DEF_AcqErr.IdXML		:=	'5';
DEF_AcqErr.TagXML		:=	7;

DEF_Prm_Pos.IdXML		:=	'5';
DEF_Prm_Pos.TagXML		:=	8;

DEF_Position.IdXML		:=	'5';
DEF_Position.TagXML		:=	1;

DEF_Rotation.IdXML		:=	'5';
DEF_Rotation.TagXML		:=	4;

DEF_Surv_rotation.IdXML	:=	'5';
DEF_Surv_rotation.TagXML:=	5;

DEF_Jog.IdXML			:=	'5';
DEF_Jog.TagXML			:=	9;

DEF_Home.IdXML			:=	'5';
DEF_Home.TagXML			:=	2;

DEF_Interlock.IdXML		:=	'0';
DEF_Interlock.TagXML		:=	5;

DEF_Asserv.IdXML		:=	'5';
DEF_Asserv.TagXML		:=	10;

DEF_Desasserv.IdXML		:=	'5';
DEF_Desasserv.TagXML	:=	11;

DEF_Reset.IdXML			:=	'5';
DEF_Reset.TagXML		:=	12;

DEF_Lag_Distance.IdXML	:=	'5';
DEF_Lag_Distance.TagXML:=	13;

DEF_Limite_Switch.IdXML	:=	'5';
DEF_Limite_Switch.TagXML:=	14;

(* réception ordres externes*)
RCP_Zero	:=	M_Zero;
RCP_Bias	:=	M_Bias;
RCP_Read_Error_Mat	:=	M_Read_Error_Mat;

(*calcul de position absolue du codeur*)
STATE_Pos_Abs_Codeur := F_ReadMotorAbsPosition(fScalingFactor := CONF_Scaling_Factor, dPositionFeedback := IN_Position_Codeur);

(*Calcul position relative + controle cohérence*)
IF OP_Position.Etape.2 OR OP_Balayage.Etape.2 OR OP_Balayage.Etape.7 OR OP_Balayage.Etape.9 THEN
	VAR_Ctrl_Cons_Ok := FALSE;
	IF ( PRM_NPoste < 0) OR (PRM_NPoste > 8) OR ( PRM_NRef < 0) OR (PRM_NRef > 8) THEN
		VAR_Ctrl_Cons_Ok := FALSE;
	ELSE
		IF (PRM_NPoste =	0) THEN
			VAR_pos_poste	:= 	0.0;
		ELSE
			VAR_pos_poste 	:= 	CONF_Pos_Poste[PRM_NPoste];
		END_IF
		IF (PRM_NRef = 0) THEN
			VAR_Pos_ref		:= 	0.0;
		ELSE
			VAR_Pos_ref		:=	CONF_Pos_Ref[PRM_Nref];
		END_IF
		VAR_cons_pos		:=	PRM_Position - Var_Pos_Poste + Var_Pos_Ref ;
		IF NOT CONF_Mvt_Lineaire THEN
			WHILE VAR_Cons_Pos > 360.0 DO
				VAR_cons_pos := VAR_cons_pos - 360;
			END_WHILE
			WHILE VAR_Cons_Pos < 0.0 DO
				VAR_cons_pos := VAR_cons_pos + 360;
			END_WHILE
			VAR_Ctrl_Cons_Ok		:=	TRUE;
		ELSE
			IF ((VAR_Cons_Pos >= CONF_Min_Pos) AND (VAR_Cons_Pos <= CONF_Max_Pos))
					OR ((CONF_Min_Pos = 0.0) AND (CONF_Max_Pos = 0.0)) THEN
				VAR_Ctrl_Cons_Ok		:=	TRUE;
			END_IF
		END_IF
	END_IF;
END_IF;

(*Calcul position par rapport au balayage*)
IF OP_Balayage.Etape.7 THEN
	VAR_Cons_Pos2 := VAR_cons_pos + PRM_Angle_Bal/2;
ELSIF OP_Balayage.Etape.9 THEN
	VAR_Cons_Pos2 := VAR_cons_pos - PRM_Angle_Bal/2;
ELSIF OP_Balayage.Etape.2 THEN
	IF NOT PRM_BalPos THEN
		VAR_Cons_Pos2 := VAR_cons_pos;
	ELSE
		VAR_Cons_Pos2 := VAR_cons_pos - PRM_Angle_Bal/2;
	END_IF
ELSIF  OP_Balayage.Etape.0 THEN
	VAR_Cons_Pos2 := VAR_cons_pos;
END_IF
IF OP_Balayage.Etape.7 OR OP_Balayage.Etape.9 OR OP_Balayage.Etape.2 OR OP_Balayage.Etape.0 THEN
	VAR_Ctrl_Cons_ok2		:=	FALSE;
	IF NOT CONF_Mvt_Lineaire THEN
		WHILE VAR_Cons_Pos2 > 360.0 DO
			VAR_Cons_Pos2 := VAR_Cons_Pos2 - 360;
		END_WHILE
		WHILE VAR_Cons_Pos2 < 0.0 DO
			VAR_Cons_Pos2 := VAR_Cons_Pos2 + 360;
		END_WHILE
		VAR_Ctrl_Cons_ok2		:=	TRUE;
	ELSE
		IF ((VAR_Cons_Pos2 >= CONF_Min_Pos) AND (VAR_Cons_Pos2 <= CONF_Max_Pos))
				OR ((CONF_Min_Pos = 0.0) AND (CONF_Max_Pos = 0.0)) THEN
			VAR_Ctrl_Cons_ok2		:=	TRUE;
		END_IF
	END_IF
END_IF

(*memorisation consigne de vitesse et conversion en deg/s si nécessaire*)
IF OP_Rotation.Etape.2 OR OP_Balayage.Etape.2 THEN
	IF CONF_Mvt_Lineaire THEN
		VAR_V_BalRot	:=	PRM_V_BalRot;
	ELSE
		VAR_V_BalRot	:=	(PRM_V_BalRot * 360) / 60;
	END_IF
END_IF;
IF CONF_Mvt_Lineaire THEN
	VAR_V_Pos			:=	PRM_V_Pos;
	VAR_V_Rattrapage	:=	CONF_V_Rattrapage;
ELSE
	VAR_V_Pos			:=	(PRM_V_Pos * 360) / 60;
	VAR_V_Rattrapage	:=	(CONF_V_Rattrapage * 360) / 60;
END_IF

(*analyse besoin rattrapage de jeu*)
IF OP_Position.Etape.6 AND CONF_Rattrapage THEN
	IF CONF_Mvt_Lineaire THEN
		VAR_Pos	:=	STATE_Pos;
	ELSIF CONF_Deploiement THEN
		VAR_Pos	:=	STATE_Pos_Dep;
	ELSE
		VAR_Pos	:=	STATE_Pos360;
	END_IF
	IF CONF_Mvt_Lineaire OR CONF_Deploiement THEN
		VAR_Rattrapage	:=	((VAR_Cons_Pos2 > VAR_Pos) AND CONF_Sens_Rattrapage)
							OR ((VAR_Cons_Pos2 < VAR_Pos) AND NOT CONF_Sens_Rattrapage);
	ELSE
		VAR_Pos		:=	VAR_Cons_Pos2 - VAR_Pos;
		WHILE VAR_Pos > 360.0 DO
			VAR_Pos := VAR_Pos - 360;
		END_WHILE
		WHILE VAR_Pos < 0.0 DO
			VAR_Pos := VAR_Pos + 360;
		END_WHILE
		VAR_Sens_Mvt	:=	(VAR_Pos < 180.0);
		VAR_Rattrapage	:=	(VAR_Sens_Mvt AND CONF_Sens_Rattrapage)
							OR (NOT VAR_Sens_Mvt AND NOT CONF_Sens_Rattrapage);
	END_IF
END_IF

(*Front montant et descendant du mode manuel*)
FD_Manual.CLK	:=	MANUAL;
FD_Manual();

(*Front  validation esclave*)
FD_Valid_Slave.CLK	:=	CO_Valid_Slave;
FD_Valid_Slave();
FP_Valid_Slave.CLK	:=	CO_Valid_Slave;
FP_Valid_Slave();

(*Couple - Mise à l'échelle*)
STATE_Torque	:=	IN_Torque / 10;
END_ACTION

END_FUNCTION_BLOCK

// ---- POUs/Composant/MVTS/FB_WritePosBias.TcPOU
FUNCTION_BLOCK FB_WritePosBias
(****************historique des versions*****************************)
(* Version 1-0 - HG - 	VERSION INIITIALE*)
(* Version 2-0 - HG - 	retour nouvelle valeur position bias
					fonction d'écriture d'une valeur de position bias données*)
(* Version 3-0 - HG - 	gestion maj position bias pour une position non nulle*)
(*************************************************************************)

(*Commande bExecute:
permet de mettre à jour le paramètre position bias de la tache NC pour que 
la position courante (IPosBias) corresponde à la position zéro (IPosZero)
la nouvelle valeur du Position Bias est renvoyée dans STATE_PosBias
*)
(*Commande bApply:
permet de mettre à jour le paramètre position bias de la tache NC
directement à une valeur donnée (IPosBias) 
*)
VAR_INPUT
	bExecute: 		BOOL;
	bApply:			BOOL;
	id: 				UINT;
	lPosBias: 		LREAL;
	IPosZero:		LREAL:=0.0;
END_VAR
VAR_OUTPUT
	bBusy: 			BOOL;
	bErr: 			BOOL;
	bDone: 			BOOL;
	STATE_PosBias:	LREAL;
END_VAR
VAR
	step: 			UINT;
	VAR_PosBias:	LREAL;
	R_TRIG0: 		R_TRIG;
	R_TRIG1: 		R_TRIG;
	ADSWRITE0: 	ADSWRITE;
	ADSREAD0:		ADSREAD;
END_VAR

CASE step OF

	0:	(*lancement*)
		R_TRIG0(CLK := bExecute);
		R_TRIG1(CLK := bApply);
		bBusy := FALSE;
		IF R_TRIG0.Q THEN
			ADSWRITE0(WRITE := FALSE);
			ADSREAD0(READ := FALSE);
			bDone := FALSE;
			bBusy := TRUE;
			bErr := FALSE;
			step := step + 1;
		END_IF
		IF R_TRIG1.Q THEN
			ADSWRITE0(WRITE := FALSE);
			ADSREAD0(READ := FALSE);
			bDone := FALSE;
			bBusy := TRUE;
			bErr := FALSE;
			step := 2;
			VAR_PosBias := lPosBias;
		END_IF

	1:	(*lecture Position bias courant*)
		ADSREAD0(
			NETID:= '',
			PORT:= 501,
			IDXGRP:= id,
			IDXOFFS:= 16#07,
			LEN:= SIZEOF(VAR_PosBias),
			DESTADDR:= ADR(VAR_PosBias),
			READ:= TRUE,
			TMOUT:= t#500ms,);
		IF NOT ADSREAD0.BUSY THEN
			IF ADSREAD0.ERR THEN
				bErr := TRUE;
				step := 0;
			ELSE
				step 			:= 	step + 1;
				VAR_PosBias	:=	VAR_PosBias - lPosBias + IPosZero;
			END_IF
		END_IF

	2:	(*écriture position bias*)
		ADSWRITE0(
			NETID:= '',
			PORT:= 501,
			IDXGRP:= id,
			IDXOFFS:= 16#07,
			LEN:= SIZEOF(VAR_PosBias),
			SRCADDR:= ADR(VAR_PosBias),
			WRITE:= TRUE,
			TMOUT:= t#500ms);
		IF NOT ADSWRITE0.BUSY THEN
			IF ADSWRITE0.ERR THEN
				bErr := TRUE;
			ELSE
				bDone := TRUE;
				STATE_PosBias	:=	VAR_PosBias;
			END_IF
			step := 0;
		END_IF

END_CASE

END_FUNCTION_BLOCK

// ---- POUs/Composant/MVTS/F_ReadMotorAbsPosition.TcPOU
FUNCTION F_ReadMotorAbsPosition : LREAL			(* Fonction qui permet de lire la position absolue du moteur à codeur absolu avec AX5000 *)
VAR_INPUT
	fScalingFactor						: LREAL;		(* facteur de mise à l'échelle, nb mm/inc voir System Manager *)
	dPositionFeedback					: DINT;			(* valeur de retour de position de l'AX5000 *)
END_VAR
VAR
	dNbTours							: DINT;			(* nombre de tours du codeur *)
	dNbInc								: DINT;			(* nombre d'inc sur le tour *)
END_VAR

dNbTours := SHR(dPositionFeedback, 20);	(* le nombre de tours est sur les 12 bits de poids fort *)
dNbInc := DINT_TO_DWORD(dPositionFeedback) AND 2#00000000000011111111111111111111;	(* le nombre d'inc est sur 20 bits *)
F_ReadMotorAbsPosition := (dNbTours * 1048576 * fScalingFactor) + (dNbInc * fScalingFactor);

END_FUNCTION

// ---- POUs/Composant/MVTS/BLOCK_MOTEUR_ATV_ETHERCAT.TcPOU
{attribute 'call_after_init'}
FUNCTION_BLOCK BLOCK_MOTEUR_ATV_ETHERCAT

(* Element rotatif consigne ana *)

(****************historique des versions*****************************)
(* Version 0-0 - HG - VERSION INIITIALE - basée sur BLOCK_MOTEUR_ATV*)
(* Version 0-1 - HG - Corrections suite débug HC*)
(*************************************************************************)

VAR_INPUT
	RESET:							BOOL;		(* Condition de réinitialisation de la fonction *)

	I_Valid_INPUT:					BOOL;		(*INPUT valide - données exploitables*)
	
	IN_WcState	 		AT %I*:		BOOL;		(*INPUT IO-link Data process*)
	IN_InfoDataState 	AT %I*:		UINT;		(*INPUT Device Slave State*)

	IN_Status			AT %I*:		UINT;		(* INPUT - Entrée statut variateur*)
	IN_Error			AT %I*:		UINT;		(* INPUT - Erreur*)
	
	OP_MVT:							BLOCK_G7;
	
	DEF_WcState:					PRCDEF;		(* Défaut données invalides - communication figée*)
	DEF_Slave:						PRCDEF;		(* Défaut esclave EtherCAT*)
	DEF_off_auto:					PRCDEF;		(* Défaut de rupture de la chaîne de sécurité*)
	DEF_Variateur:					PRCDEF;		(* Défaut indiquant que le variateur n'est pas ok*)

	PRM_Vitesse:					REAL;		(* Consigne vitesse moteur*)
	PRM_Rapport:					REAL;		(* Rapport chaine cinématique*)
	
	CO_On:							BOOL;		(* Marche moteur en automatique*)
END_VAR

VAR_OUTPUT
	OUT_Control		AT %Q*:			UINT;		(* OUTPUT - Sortie mode de controle*)
	OUT_Velocity	AT %Q*:			INT;		(* OUTPUT - Sortie consigne vitesse, attention sortie en rpm ex: moteur a Vnom 1500 rpm*)

	STATE_Ready:					BOOL; 		(* Moteur pret*)
	STATE_OFF:						BOOL;		(* Moteur à l'arrêt *)
	STATE_EC:						BOOL;		(* Asservissement en cours *)
	STATE_ON:						BOOL;		(* Moteur en marche  *)
	STATE_NOK:						BOOL;		(* Moteur en defaut  *)
	STATE_VIT:						REAL;		(* Vitesse appliquée *)
END_VAR

VAR
	VAR_Valid_Elmt:					BOOL;		(*données EtherCAT exploitables*)

	VAR_On:							BOOL;		(* variable intermédiaire de marche moteur*)
	
	VAR_IN_ReadyToSwitchOn:			BOOL;		(* En attente de l'alimentation de puissance=1*)
	VAR_IN_SwitchedOn:				BOOL;		(*Ready*)
	VAR_IN_OperationEnabled:		BOOL;		(*En fonctionnement*)
	VAR_IN_Fault:					BOOL;		(* error*)
	VAR_IN_VoltageEnabled:			BOOL;		(*Alim puissance présente *)
	VAR_IN_QuickStop:				BOOL;		(* Arret rapide =0*)		
	VAR_IN_SwitchOnDisabled:		BOOL;		(* Absence Alim puissance *)
	VAR_IN_Warning:					BOOL;		(* Alarme présente*)
	VAR_IN_Reserve1:				BOOL;
	VAR_IN_Remote:					BOOL;		(* Commande via bus de terrain*)
	VAR_IN_TargetReached:			BOOL;		(* Référence atteinte*)
	VAR_IN_InternalLimitActive:		BOOL;		(* Déppassement réf*)
	VAR_IN_Reserve2:				BOOL;
	VAR_IN_Reserve3:				BOOL;
	VAR_IN_Conf1:					BOOL;		(* Stop button*)
	VAR_IN_Conf2:					BOOL;		(*Sens de rotations*)
	VAR_Status_Code:				USINT;		(*1: not ready to switch on, 2: switch on disabled, 3: ready to switch on,
												4: switched on, 5: operation enabled, 6: quick stop active,
												7: fault reaction active, 8: fault*)														
	VAR_OUT_SwitchOn:				BOOL;		(*Contrôle du switch principal*)
	VAR_OUT_EnableVoltage:			BOOL;		(*Mise en puissance*)
	VAR_OUT_QuickStop:				BOOL;		(*Quick stop activé =0*)
	VAR_OUT_EnableOperation:		BOOL;		(*Commande activée =1*)
	VAR_OUT_Reserve1:				BOOL;
	VAR_OUT_Reserve2:				BOOL;
	VAR_OUT_Reserve3:				BOOL;
	VAR_OUT_FaultReset:				BOOL;		(*0 à 1 pour reset erreur si l'erreur n'est plus active*)
	VAR_OUT_Halt:					BOOL;		(*0= run demandé, 1=arrêt demandé*)
	VAR_OUT_Reserve4:				BOOL;
	VAR_OUT_Reserve5:				BOOL;
	VAR_OUT_Conf1:					BOOL;		(*C311 - Marche avant par défaut*)  (*0= Marche avant demandée, 1= marche arrière demandée*)
	VAR_OUT_Conf2:					BOOL;		(*C312 - Marche arrière par défaut*)
	VAR_OUT_Conf3:					BOOL;		(*C313*)
	VAR_OUT_Conf4:					BOOL;		(*C314*)
	VAR_OUT_Conf5:					BOOL;		(*C315*)
	
	TIMER_Reset:					TON;
	TIMER_Timeout_Fault:			TON;
END_VAR

VAR_INPUT PERSISTENT
	CONF_VMAX:					REAL;			(*Consigne vitesse max*)
	CONF_VMIN:					REAL;			(*Consigne vitesse min*)
	CONF_No_Safety_Auto:		BOOL:=FALSE;	(*Option de desactivation des conditions d'autorisation en mode automatique*)
	
	(*Entité*)
	IsComponent:		BOOL;			(*entité : assembly*)
	IdXML:			STRING;			(*nom entité : identifiant pour recherche dans dico*)
	TagXML:			UINT;			(*nom entité : identifiant pour recherche dans dico*)
	IdParent:			STRING;			(*MNEMO de l'appelant*)
	MNEMO:			STRING;			(*MNEMO de l'entité*)
END_VAR

IdXML:= '5';
TagXML:= 2;

DEF_OFF_AUTO.IdXML := '3';
DEF_OFF_AUTO.TagXML :=10;
DEF_Variateur.IdXML	:= '5';
DEF_Variateur.TagXML:= 15;
DEF_Slave.IdXML := '19';
DEF_Slave.TagXML := 2;
DEF_WcState.IdXML := '19';
DEF_WcState.TagXML := 1;

(*DEFAUTS ESCLAVE ETHERCAT*)
(*Défaut données invalides*)
DEF_WcState.CONDITION	:=	IN_WcState AND NOT I_Valid_INPUT;
DEF_WcState();
(*Défaut esclave etherCAT*)
DEF_Slave.CONDITION		:=	(IN_InfoDataState<>8) AND NOT I_Valid_INPUT;
DEF_Slave.VAL1			:=	UINT_TO_STRING(IN_InfoDataState);
DEF_Slave();

(*Données E/S valables*)
VAR_Valid_Elmt			:=	I_Valid_INPUT AND NOT DEF_WcState.DEF AND NOT DEF_Slave.DEF;

(*Réception status*)
VAR_IN_ReadyToSwitchOn		:=	IN_Status.0;
VAR_IN_SwitchedOn			:=	IN_Status.1;
VAR_IN_OperationEnabled		:=	IN_Status.2;
VAR_IN_Fault				:=	IN_Status.3;
VAR_IN_VoltageEnabled		:=	IN_Status.4;
VAR_IN_QuickStop			:=	IN_Status.5;
VAR_IN_SwitchOnDisabled		:=	IN_Status.6;
VAR_IN_Warning				:=	IN_Status.7;
VAR_IN_Reserve1				:=	IN_Status.8;
VAR_IN_Remote				:=	IN_Status.9;
VAR_IN_TargetReached		:=	IN_Status.10;
VAR_IN_InternalLimitActive	:=	IN_Status.11;
VAR_IN_Reserve2				:=	IN_Status.12;
VAR_IN_Reserve3				:=	IN_Status.13;
VAR_IN_Conf1				:=	IN_Status.14;
VAR_IN_Conf2				:=	IN_Status.15;

(*CODE STATUS*)
IF NOT VAR_IN_ReadyToSwitchOn AND NOT VAR_IN_SwitchedOn AND NOT VAR_IN_OperationEnabled AND NOT VAR_IN_Fault AND NOT VAR_IN_SwitchOnDisabled THEN
	VAR_Status_Code	:=	1;	(*Not ready to switch on*)
ELSIF NOT VAR_IN_ReadyToSwitchOn AND NOT VAR_IN_SwitchedOn AND NOT VAR_IN_OperationEnabled AND NOT VAR_IN_Fault AND VAR_IN_SwitchOnDisabled THEN
	VAR_Status_Code	:=	2;	(*Switch on disabled*)
ELSIF VAR_IN_ReadyToSwitchOn AND NOT VAR_IN_SwitchedOn AND NOT VAR_IN_OperationEnabled AND NOT VAR_IN_Fault AND VAR_IN_QuickStop AND NOT VAR_IN_SwitchOnDisabled THEN
	VAR_Status_Code	:=	3;	(*Ready to switch on*)
ELSIF VAR_IN_ReadyToSwitchOn AND VAR_IN_SwitchedOn AND NOT VAR_IN_OperationEnabled AND NOT VAR_IN_Fault AND VAR_IN_VoltageEnabled AND VAR_IN_QuickStop AND NOT VAR_IN_SwitchOnDisabled THEN
	VAR_Status_Code	:=	4;	(*Switched on*)
ELSIF VAR_IN_ReadyToSwitchOn AND VAR_IN_SwitchedOn AND VAR_IN_OperationEnabled AND NOT VAR_IN_Fault AND VAR_IN_VoltageEnabled AND VAR_IN_QuickStop AND NOT VAR_IN_SwitchOnDisabled THEN
	VAR_Status_Code	:=	5;	(*Operation enabled*)
ELSIF VAR_IN_ReadyToSwitchOn AND VAR_IN_SwitchedOn AND VAR_IN_OperationEnabled AND NOT VAR_IN_Fault AND VAR_IN_VoltageEnabled AND NOT VAR_IN_QuickStop AND NOT VAR_IN_SwitchOnDisabled THEN
	VAR_Status_Code	:=	6;	(*Quick stop active*)
ELSIF VAR_IN_ReadyToSwitchOn AND VAR_IN_SwitchedOn AND VAR_IN_OperationEnabled AND VAR_IN_Fault AND NOT VAR_IN_SwitchOnDisabled THEN
	VAR_Status_Code	:=	7;	(*Fault reaction active*)
ELSIF NOT VAR_IN_ReadyToSwitchOn AND NOT VAR_IN_SwitchedOn AND NOT VAR_IN_OperationEnabled AND VAR_IN_Fault AND NOT VAR_IN_SwitchOnDisabled THEN
	VAR_Status_Code	:=	8;	(*Fault*)
END_IF


(*Vérification consignes*)
IF	PRM_Vitesse > CONF_VMAX THEN
	PRM_Vitesse	:=	CONF_VMAX;
END_IF;

IF PRM_Vitesse < CONF_VMIN THEN
	PRM_Vitesse := CONF_VMIN;
END_IF


(*défaut desactivation automatique*)
DEF_off_auto.CONDITION	:=	(DEF_Variateur.DEF AND NOT OP_MVT.Etape.1 AND NOT OP_MVT.Etape.2 AND NOT OP_MVT.Etape.0)
							OR TIMER_Timeout_Fault.Q;
DEF_off_auto.DELAY		:=	T#0MS;
DEF_off_auto();

(*défaut du variateur*)
DEF_Variateur.CONDITION		:= 	VAR_IN_Fault OR VAR_IN_Warning;
DEF_Variateur.VAL1			:=	UINT_TO_STRING(IN_Error);
DEF_Variateur.DELAY			:= 	T#5MS;
DEF_Variateur();

(*Indicateur prêt*)
STATE_Ready		:=	VAR_Valid_Elmt;

(*gestion des sorties*)
VAR_On		:= 	CO_ON AND NOT RESET;

(*appel G7*)
ACT_MVT();


(*consigne vitesse*)
IF	STATE_ON AND (PRM_VITESSE<>STATE_VIT) THEN
	OUT_Velocity	:=	REAL_TO_INT(PRM_Vitesse*PRM_Rapport);
	STATE_VIT		:=	PRM_Vitesse;
ELSIF STATE_OFF THEN
	OUT_Velocity	:=	0;
	STATE_VIT		:=	0;
END_IF;

(*PILOTAGE MODE DE CONTROLE*)
VAR_OUT_Conf1		:=	FALSE;
VAR_OUT_Conf2		:=	FALSE;
VAR_OUT_Conf3		:=	FALSE;
VAR_OUT_Conf4		:=	FALSE;
VAR_OUT_Conf5		:=	FALSE;
VAR_OUT_Reserve1	:=	FALSE;
VAR_OUT_Reserve2	:=	FALSE;
VAR_OUT_Reserve3	:=	FALSE;
VAR_OUT_Reserve4	:=	FALSE;
VAR_OUT_Reserve5	:=	FALSE;

VAR_OUT_Halt		:=	FALSE;

VAR_OUT_FaultReset		:=	OP_MVT.Etape.2;
VAR_OUT_EnableVoltage	:=	OP_MVT.Etape.3 OR OP_MVT.Etape.4 OR OP_MVT.Etape.5 OR OP_MVT.Etape.6 OR OP_MVT.Etape.7;
VAR_OUT_SwitchOn		:=	OP_MVT.Etape.4 OR OP_MVT.Etape.5 OR OP_MVT.Etape.6 OR OP_MVT.Etape.7;
VAR_OUT_QuickStop		:=	OP_MVT.Etape.3 OR OP_MVT.Etape.4 OR OP_MVT.Etape.5 OR OP_MVT.Etape.6 OR OP_MVT.Etape.7;
VAR_OUT_EnableOperation	:=	OP_MVT.Etape.5 OR OP_MVT.Etape.6;
//VAR_OUT_Conf1			:=	OP_MVT.Etape.6 AND (PRM_Vitesse > 0.0);

//MEMCPY(ADR(OUT_Control),ADR(VAR_OUT_SwitchOn),16);
OUT_CONTROL.0:=VAR_OUT_SwitchOn;
OUT_CONTROL.1:=VAR_OUT_EnableVoltage;
OUT_CONTROL.2:=VAR_OUT_QuickStop;
IdXML:= '5';
TagXML:= 2;

DEF_OFF_AUTO.IdXML := '3';
DEF_OFF_AUTO.TagXML :=10;
(*DEF_MARCHE.IdXML := '3';
DEF_MARCHE.TagXML:=1;*)
DEF_Variateur.IdXML	:= '5';
DEF_Variateur.TagXML:= 15;
	
	
OUT_CONTROL.3:=VAR_OUT_EnableOperation;
OUT_CONTROL.4:=VAR_OUT_Reserve1;
OUT_CONTROL.5:=VAR_OUT_Reserve2;
OUT_CONTROL.6:=VAR_OUT_Reserve3;
OUT_CONTROL.7:=VAR_OUT_FaultReset;
OUT_CONTROL.8:=VAR_OUT_Halt;
OUT_CONTROL.9:=VAR_OUT_Reserve4;
OUT_CONTROL.10:=VAR_OUT_Reserve5;
OUT_CONTROL.11:=VAR_OUT_Conf1;
OUT_CONTROL.12:=VAR_OUT_Conf2;
OUT_CONTROL.13:=VAR_OUT_Conf3;
OUT_CONTROL.14:=VAR_OUT_Conf4;
OUT_CONTROL.15:=VAR_OUT_Conf5;


(*Gestion du TIMER RESET*)
Timer_reset.IN:=OP_MVT.Etape.2;
Timer_reset.PT:= T#2S;
Timer_reset();

(*Gestion du TIMER Timout reset*)
TIMER_Timeout_Fault.IN:=OP_MVT.Etape.1 OR OP_MVT.Etape.2;
TIMER_Timeout_Fault.PT:=T#7S;
TIMER_Timeout_Fault();

(*Indicateur defaut*)
STATE_NOK	:=	DEF_off_auto.DEF OR DEF_Variateur.DEF OR DEF_WcState.DEF OR DEF_Slave.DEF;
STATE_ON	:=	OP_MVT.Etape.6;
STATE_OFF	:=	OP_MVT.Etape.0;
STATE_EC	:=	NOT STATE_ON AND NOT STATE_OFF;

ACTION ACT_MVT:
OP_MVT(
	N_STEP_OP_OK:= 6,
	N_STEP_OP_NOK:= 0);

(*GRAFCET*)
(* initialisation du grafcet*)
IF 		OP_MVT.ETAPE = 0
		THEN
				OP_MVT.ETAPE.0 := TRUE;
(*repositionnement sur étape 0*)
ELSIF	(NOT VAR_On OR DEF_off_auto.DEF)
		AND NOT OP_MVT.Etape.6 AND NOT OP_MVT.Etape.7
		THEN
				OP_MVT.ETAPE := 0;			(*RAZ grafcet*)
				OP_MVT.ETAPE.0:=TRUE;
(*étape 0-1*)
ELSIF 	OP_MVT.ETAPE.0
		AND VAR_On
		THEN
				OP_MVT.ETAPE.1:=TRUE;
				OP_MVT.ETAPE.0:=FALSE;
(*étape 1-2 : Fault*)
ELSIF	OP_MVT.Etape.1
		AND (VAR_Status_Code = 8)
		THEN
				OP_MVT.ETAPE.2:=TRUE;
				OP_MVT.ETAPE.1:=FALSE;
(*étape 2-1 : reset fault*)
ELSIF	OP_MVT.Etape.2
		AND TIMER_Reset.Q
		THEN
				OP_MVT.ETAPE.1:=TRUE;
				OP_MVT.ETAPE.2:=FALSE;				
(*étape 1-3*)
ELSIF	OP_MVT.Etape.1
		AND (VAR_Status_Code >= 2)
		THEN
				OP_MVT.ETAPE.3:=TRUE;
				OP_MVT.ETAPE.1:=FALSE;		
(*étape 3-4*)
ELSIF	OP_MVT.Etape.3
		AND (VAR_Status_Code >= 3)
		THEN
				OP_MVT.ETAPE.4:=TRUE;
				OP_MVT.ETAPE.3:=FALSE;	
(*étape 4-5*)
ELSIF	OP_MVT.Etape.4
		AND (VAR_Status_Code = 4)
		THEN
				OP_MVT.ETAPE.5:=TRUE;
				OP_MVT.ETAPE.4:=FALSE;
(*étape 5-6*)
ELSIF	OP_MVT.Etape.5
		AND (VAR_Status_Code = 5)
		THEN
				OP_MVT.ETAPE.6:=TRUE;
				OP_MVT.ETAPE.5:=FALSE;
(*étape 6-7*)
ELSIF	OP_MVT.Etape.6
		AND (NOT VAR_On OR DEF_off_auto.DEF)
		THEN
				OP_MVT.ETAPE.7:=TRUE;
				OP_MVT.ETAPE.6:=FALSE;
(*étape 7-0*)
ELSIF	OP_MVT.Etape.7
		AND (VAR_Status_Code <> 5)
		THEN
				OP_MVT.ETAPE.0:=TRUE;
				OP_MVT.ETAPE.7:=FALSE;
END_IF

OP_MVT.POST();
END_ACTION

END_FUNCTION_BLOCK

// ---- POUs/Composant/POMPES/BLOCK_PPM_DEF.TcPOU
FUNCTION_BLOCK BLOCK_PPM_DEF

(* Gestion d'une pompe turbo ADIXEN avec controleur REMOTE*)
(* TYPE OBJET = POMPE TURBO*)

(****************historique des versions*****************************)

(* Version 1-0 - HG - VERSION INIITIALE - 7015*)
(* Version 2-0 - HG - 06/2011 - Adaptation pour journal des évènements externe*)

(*************************************************************************)

VAR_INPUT
	MANUAL:					BOOL;				(* Mode de pilotage manuel *)
	RESET:					BOOL;				(* Condition de réiinitialisation de la fonction *)
	WATER:					BOOL;				(*indication de refrodissement de la pompe ok*)

	DEF_Arret_Auto:			PRCDEF;		(*01 - défaut d'arrêt automatique de la pompe*)
	DEF_Marche_imposs:		PRCDEF;		(*02 - défaut de marche de la pompe turbo non autorisée*)
	DEF_Arret_imposs:		PRCDEF;		(*03 - défaut d'arrêt de la pompe turbo non autorisée*)
	DEF_On:					PRCDEF;		(*04 - défaut de marche de la pompe*)
	DEF_Off:				PRCDEF;		(*05 - défaut d'arrêt de la pompe*)
	DEF_Interne:			PRCDEF;		(*06 - défaut interne de la pompe*)

	CO_On:					BOOL;			(*demande de marche de la pompe en mode automatique généré par la fonction qui gère la pompe*)

	(*conditions d'autorisation*)
	EN_On_INT:					BOOL:= TRUE;	(*condition d'autorisation de marche et de standby de la pompe donnée par la fonction qui gère la pompe*)
	EN_Off_INT:					BOOL:= TRUE;	(*condition d'autorisation d'arrêt de la pompe donnée par la fonction qui gère la pompe*)
	EN_On_EXT:					BOOL:= TRUE;	(*condition d'autorisation de marche et de standby externe*)
	EN_Off_EXT:					BOOL:= TRUE;	(*condition d'autorisation d'arrêt de la pompe donnée par la fonction qui gère la pompe*)

	IN_On:						BOOL;			(*entrée TOR pompe en marche*)
	IN_Def:						BOOL;			(*entrée TOR pompe en défaut*)

	OUT_On:						BOOL;			(* Marche pompe *)
END_VAR

VAR_INPUT PERSISTENT
	CONF_Tim_Valid_On:			TIME:=T#0ms;	(*temporisation de validation du l'état STATE_OK*)
	CONF_Tim_Valid_Off:			TIME:=T#0ms;	(*temporisation de validation de l'état STATE_AR*)

	(*Entité*)
	IsComponent:		BOOL;			(*entité : composant*)
	IdXML:				STRING;			(*nom entité : identifiant pour recherche dans dico*)
	TagXML:				UINT;			(*nom entité : identifiant pour recherche dans dico*)
	IdParent:			STRING;			(*MNEMO de l'appelant*)
	MNEMO:				STRING;			(*MNEMO de l'entité*)
END_VAR

VAR_OUTPUT
	RQ_Cool:					BOOL;			(* Demande de refroidissement de la pompe turbo*)

	(*variable d'état d'autorisation*)
	AUTOR_On_IHM:				BOOL;			(*indique que la mise en marche de la pompe est autorisée en mode manuel depuis l'IHM*)
	AUTOR_Off_IHM:				BOOL;			(*indique que l'arrêt de la pompe est autorisée en mode manuel depuis l'IHM*)

	STATE_Ec:					BOOL;			(*indique que la pompe est en marche et n'a pas atteint sa vitesse*)
	STATE_On:					BOOL;			(*indique que la pompe est en marche et à atteint sa vitesse*)
	STATE_NOK:					BOOL;			(*indique la présence d'un défaut sur la pompe ou que l'ordre de marche a été refusé*)
	STATE_Off:					BOOL;			(*indique que la pompe est à l'arrêt*)
	STATE_Ihm:					USINT;			(*code d'état de la pompe*)
END_VAR

VAR
	TIMER_Valid_On:				TON;
	TIMER_Valid_Off:			TON;

	(* Variables demande en mode manuel*)
	M_On:						BOOL;			(* Ordre marche/arrêt de la  pompe en mode manuel *)
	RCP_M_On:					BOOL;			(* bit de reception de l'ordre de marche en mode manuel*)
	VAR_On:						BOOL;			(* variable intermédiaire de marche de la pompe*)

	VAR_CPT:					BLOCK_CPT_TEMPS;
END_VAR

VAR_EXTERNAL
	MANUAL_SAFETY_OFF:			BOOL;			(*desactive les sécurités en mode manuel*)
END_VAR

DEF_Arret_Auto.IdXml			:=	'3';
DEF_Arret_Auto.TagXml			:=	10;

DEF_Marche_imposs.IdXml			:=	'3';
DEF_Marche_imposs.TagXml		:=	5;

DEF_Arret_imposs.IdXml			:=	'3';
DEF_Arret_imposs.TagXml			:=	8;

DEF_On.IdXml					:=	'3';
DEF_On.TagXml					:=	1;

DEF_Off.IdXml					:=	'3';
DEF_Off.TagXml					:=	3;

DEF_Interne.IdXml				:=	'0';
DEF_Interne.TagXml				:=	6;


(* Gestion des ordres en mode manuel *)
RCP_M_On 				:=	M_On;

(*gestion des bits d'autorisation en mode manuel*)
AUTOR_On_IHM			:=	NOT RESET AND ((EN_On_INT AND EN_On_EXT AND WATER AND NOT DEF_Interne.DEF) OR MANUAL_SAFETY_OFF)
							AND NOT VAR_On  AND MANUAL;
AUTOR_Off_IHM			:=	NOT RESET  AND VAR_On  AND MANUAL
							AND (( EN_Off_EXT AND EN_Off_INT) OR MANUAL_SAFETY_OFF);

(*défaut d'arrêt automatique de la pompe *)
DEF_Arret_Auto.CONDITION :=     (NOT WATER
								OR  NOT EN_On_INT
								OR NOT EN_On_EXT
								OR DEF_Interne.DEF)
								AND  OUT_On AND NOT RESET;
DEF_arret_auto.DELAY:=T#0ms;
DEF_Arret_Auto();

(* Défaut de marche de la pompe primaire non autorisée en automatique*)
DEF_marche_imposs.CONDITION:=	NOT MANUAL AND CO_On AND (NOT EN_On_INT OR NOT EN_On_EXT)
								AND NOT MANUAL AND NOT RESET;
DEF_marche_imposs.DELAY := T#0ms;
DEF_marche_imposs();

(* Défaut d'arrêt de la pompe primaire non autorisée en automatique*)
DEF_arret_imposs.CONDITION	:=	NOT MANUAL AND NOT CO_On AND VAR_ON AND( NOT EN_Off_INT OR NOT EN_Off_EXT)
								AND NOT RESET;
DEF_arret_imposs.DELAY := T#0ms;
DEF_arret_imposs();

(* ARRET POMPE*)
IF 		(NOT CO_On AND NOT MANUAL AND EN_Off_INT AND EN_Off_EXT)
		OR ( RCP_M_On AND AUTOR_Off_IHM) OR RESET OR DEF_arret_auto.DEF
		THEN
			Var_On 				:= 	FALSE;
(*MARCHE POMPES*)
ELSIF	( CO_On AND NOT MANUAL AND EN_On_INT AND EN_On_EXT)
		 OR 	( RCP_M_On AND AUTOR_On_IHM) THEN
			Var_On 				:= 	TRUE;
END_IF;

(*SORTIE MARCHE POMPE*)
OUT_On			:= 	WATER AND VAR_On;

(*DEMANDE DE REFROIDISSEMENT DE LA POMPE*)
RQ_Cool			:=	VAR_On;

(* Défaut de marche de la pompe*)
DEF_ON.CONDITION := OUT_On AND NOT IN_On;
DEF_ON();

(* Défaut d'arrêt de la pompe*)
DEF_Off.CONDITION := NOT OUT_On AND IN_On;
DEF_Off();

(*Défaut interne de la pompe*)
DEF_Interne.CONDITION := IN_Def;
DEF_Interne.DELAY :=	T#200ms;
DEF_Interne();

(*affectation des bits d'état*)
(*indicateur pompe en marche STATE_ON*)
TIMER_Valid_On.IN	:=	OUT_On AND IN_On;
TIMER_Valid_On(PT:=CONF_Tim_Valid_On);
STATE_ON			:=	TIMER_Valid_On.Q;
(*indicateur pompe à l'arrêt STATE_OFF*)
TIMER_Valid_Off.IN	:=	NOT OUT_On AND NOT IN_On;
TIMER_Valid_Off(PT:=CONF_Tim_Valid_Off);
STATE_Off			:=	TIMER_Valid_Off.Q;
	STATE_Ec		:=	VAR_On AND NOT IN_On;
	STATE_NOK		:=	DEF_Arret_imposs.DEF OR DEF_Marche_imposs.DEF OR DEF_Arret_auto.DEF OR DEF_On.DEF OR DEF_Off.DEF OR DEF_Interne.DEF;

IF NOT out_on THEN
	STATE_Ihm := 0;
ELSIF out_on AND NOT IN_On THEN
	STATE_ihm := 1;
ELSIF out_on AND in_on THEN
	STATE_ihm:=2;
END_IF;


(*Gestion compteur*)
VAR_CPT(I_On:= STATE_On);

(* Reset des ordres*)
	IF M_On AND RCP_M_On THEN
		M_On		:= FALSE;
	END_IF;

END_FUNCTION_BLOCK

// ---- POUs/Composant/POMPES/BLOCK_PTM_OBCV4.TcPOU
FUNCTION_BLOCK BLOCK_PTM_OBCV4

(****************historique des versions************************************)

(* Version 1-0 - ?? - ??/?? -  VERSION INIITIALE*)
(* Version 2-0 - HG - 02/2013 - Adaptation pour journal des évènements externe, renommage variables*)
(* Version 2-1 - GV - 10/2017 - Gestion arrêt automatique *)

(********************************************************************************)

VAR_INPUT
	EN_On_EXT:				BOOL;	(* Autorisation de marche en mode manuel *)
	EN_Off_EXT:				BOOL;	(* Autorisation d'arrêt en mode manuel *)
	EN_On_INT:				BOOL;
	EN_Off_INT:				BOOL;

	EN_Purge_EXT:			BOOL;	(*Autorisation externe d'ouverture de la vanne de purge : typiquement, VI en amont de PS ouverte*)

	CO_On:					BOOL;	(* Ordre automatique de marche pompe *)
	CO_Purge:				BOOL;	(* Ordre automatique d'ouverture de la vanne de purge de la pompe (pas de gestion manuelle de cette vanne)*)

	MANUAL:					BOOL;	(* Ordre de commande manuel de la fonction *)
	RESET: 					BOOL;	(* Condition de réiinitialisation de la fonction *)
	WATER:					BOOL;	(* Indication de refrodissement de la pompe ok*)
	I_Standby:				BOOL;	(* Condition réduction vitesse pompe *)

	DEF_Arret_Auto:			PRCDEF;	(* Indicateur de défaut d'arrêt automatique de la pompe*)
	DEF_On:					PRCDEF;	(* Indicateur de défaut amorçage de la pompe turbo *)
	DEF_Off:				PRCDEF;	(* Indicateur de défaut d'arrêt de la pompe turbo *)
	DEF_Desamorcage:		PRCDEF;	(* Indicateur de défaut désamorçage de la pompe turbo *)
	DEF_Interne:			PRCDEF;	(* Indicateur de défaut interne de la pompe turbo *)
	DEF_Marche_Imposs:		PRCDEF;	(* Indicateur de défaut de marche de la pompe turbo non autorisée*)
	DEF_Arret_Imposs:		PRCDEF;	(* Indicateur de défaut d'arrêt de la pompe turbo non autorisée*)
END_VAR

VAR_OUTPUT
	STATE_Erreur:			INT;			(* Code erreur du défaut interne de la pompe *)
	RQ_Cool:				BOOL;
	Autor_ON_IHM:			BOOL;
	Autor_Off_IHM:			BOOL;
END_VAR

VAR
	INPUT1	AT %I*:		USINT;
	OUTPUT1	AT%Q*:		USINT;

	(* Variables pour l'entrée profibus *)
	STATE_On:				BOOL;		(* Normal operation has been attained *)
	STATE_Off:				BOOL;		(* Pump is off *)
	STATE_NOK:				BOOL;
	VAR_Ok:					BOOL;		(* pump at speed *)
	VAR_PSxM_ec:			BOOL;		(* Pump is running *)
	VAR_Maint_required:		BOOL;		(* Maintenance is required *)
	VAR_Error_active:		BOOL;		(* Error active *)
	VAR_Com_int_fault:		BOOL;		(* Internal communication failure *)
	VAR_Overbalance_fault:	BOOL;		(* Overbalance default *)
	VAR_Overtemp_pump_fault:BOOL;		(* Overtemperature pump warning *)
	VAR_Overtemp_ctrl_fault:BOOL;		(* Overtemperature controller warninq *)

	(* Variables pour les sorties profibus *)
	VAR_PSx:				BOOL;		(* Start pump *)
	VAR_Enable_process:		BOOL;		(* Enable process data *)
	VAR_Purge_gaz_on:		BOOL;		(* Purge gaz valve on *)
	VAR_Foreline_isol_on:	BOOL;		(* Foreline isolation valve on *)
	VAR_Standby_speed:		BOOL;		(* Go to standby speed *)
	VAR_Ack_error:			BOOL;		(* Acknowledge error *)

	(* Variables pour IHM *)
	M_ON:					BOOL;		(* Ordre maintenance commutation sortie marche pompe *)
	RCP_M_PSx:				BOOL;

	(* Variables interne à la fonction *)
	FD_PSxM:				F_TRIG;

	TIMER_Valid_On:			TON;
	TIMER_Valid_Off:		TON;

END_VAR

VAR_INPUT PERSISTENT
	(*Entité*)
	IsComponent:			BOOL;			(*entité : composant*)
	IdXML:					STRING;			(*nom entité : identifiant pour recherche dans dico*)
	TagXML:					UINT;			(*nom entité : identifiant pour recherche dans dico*)
	IdParent:				STRING;			(*MNEMO de l'appelant*)
	MNEMO:					STRING;			(*MNEMO de l'entité*)
	(*parametre de configuration constructeur*)
	(*les parametres suivants dépendent de la configuration de la machine*)
	CONF_No_Safety_Auto:	BOOL:=FALSE;	(*option de desactivation des conditions d'autorisation en mode automatique*)
	CONF_Tim_Valid_On:  	TIME; 			(*Temps validation actionneur on*)
	CONF_Tim_Valid_Off:   	TIME; 			(*Temps validation actionneur off *)
END_VAR

(*Gestion d'une pompe turbo indépendante
La fonction permet de gérer la mise en CO_On de la pompe  sur une 
condition et l'arrêt  sur la remise à 0 de la condition de CO_On en mode 
automatique
La fonction gère des défauts d'amorçage et de désamorçage  et la commutation de 
l'état de la pompe en mode maintenance.
Défaut interne:
1:maintenance demandée, 2:communication interne, 3:équilibrage, 4:surchauffe 
pompe, 5:surchauffe controleur *)

IdXML							:=	'1';
TagXML							:=	8;

DEF_Arret_Auto.IdXml			:=	'3';
DEF_Arret_Auto.TagXml			:=	10;

DEF_Arret_imposs.IdXml			:=	'3';
DEF_Arret_imposs.TagXml			:=	8;

DEF_Off.IdXml					:=	'3';
DEF_Off.TagXml					:=	3;

DEF_On.IdXml					:=	'3';
DEF_On.TagXml					:=	1;

DEF_Marche_imposs.IdXml			:=	'3';
DEF_Marche_imposs.TagXml		:=	5;

DEF_Desamorcage.IdXml			:=	'1';
DEF_Desamorcage.TagXml			:=	13;

DEF_Interne.IdXml				:=	'0';
DEF_Interne.TagXml				:=	6;

(* Reception trame *)
VAR_Ok						:=	INPUT1.0;
VAR_PSxM_ec					:= 	INPUT1.1;
VAR_Maint_required			:=	INPUT1.2;
VAR_Error_active			:=	INPUT1.3;
VAR_Com_int_fault			:=	INPUT1.4;
VAR_Overbalance_fault 		:=	INPUT1.5;
VAR_Overtemp_pump_fault		:=	INPUT1.6;
VAR_Overtemp_ctrl_fault		:=	INPUT1.7;

(* Gestion des ordres de CO_On externe *)
RCP_M_PSx := M_ON;

(* AFFECTATION DES SORTIES LOGIQUES *)
(* state on *)
TIMER_Valid_On.PT	:=	CONF_Tim_Valid_On;
TIMER_Valid_On.IN	:=	VAR_Ok;
TIMER_Valid_On();
STATE_On			:=	TIMER_Valid_On.Q;

(* Autorisation *)
(*gestion des bits d'autorisation en mode manuel*)
AUTOR_On_IHM			:=	NOT RESET AND ((EN_On_INT AND EN_On_EXT AND WATER) OR MANUAL_SAFETY_OFF)
							AND NOT VAR_PSx  AND MANUAL;
AUTOR_Off_IHM			:=	NOT RESET  AND VAR_PSx  AND MANUAL
							AND (( EN_Off_EXT AND EN_Off_INT) OR MANUAL_SAFETY_OFF);

IF EN_On_EXT = TRUE OR EN_Off_EXT = TRUE THEN
	VAR_Enable_process :=TRUE;
ELSE
	VAR_Enable_process :=FALSE;
END_IF

(* PSx *)
IF (EN_Off_INT AND NOT CO_On AND NOT MANUAL)
		OR (STATE_On AND (RCP_M_PSx AND (EN_Off_EXT OR CONF_No_Safety_Auto) OR NOT EN_On_EXT AND MANUAL))
		OR RESET OR DEF_Arret_Auto.DEF THEN
	VAR_PSx := FALSE;
ELSIF (RCP_M_PSx AND MANUAL AND (EN_On_EXT OR CONF_No_Safety_Auto) AND NOT VAR_PSx)
		OR (WATER AND CO_On AND NOT MANUAL AND EN_On_INT) THEN
	VAR_PSx := TRUE;
END_IF

(* standby *)
IF VAR_PSx AND STATE_On AND I_Standby THEN
	VAR_Standby_speed := TRUE;
ELSE
	VAR_Standby_speed := FALSE;
END_IF

(*Purge : demande de purge externe ou phase de ralentissement de la pompe*)
VAR_Purge_gaz_on	:=	( (CO_Purge AND NOT RESET) OR (NOT VAR_PSx AND VAR_PSxM_ec) )
						AND EN_Purge_EXT;

(* state off  *)
TIMER_Valid_Off.PT	:=	CONF_Tim_Valid_Off;
TIMER_Valid_Off.IN	:=	NOT STATE_On AND NOT VAR_PSxM_ec;
TIMER_Valid_Off();
STATE_Off			:=	TIMER_Valid_Off.Q;

RQ_Cool		:=	VAR_PSx;

(* Envoi trame *)
OUTPUT1.0	:=	VAR_PSx;
OUTPUT1.2	:=	VAR_Enable_process;
OUTPUT1.4	:=	VAR_Purge_gaz_on;
OUTPUT1.5	:=	VAR_Foreline_isol_on;
OUTPUT1.6	:=	VAR_Standby_speed;
OUTPUT1.7	:=	VAR_Ack_error;

(* Défaut *)

(* Défaut de marche de la pompe primaire non autorisée en automatique*)
DEF_Marche_Imposs.CONDITION	:=	NOT MANUAL AND CO_On AND (NOT EN_On_INT OR NOT EN_On_EXT)
									AND NOT MANUAL AND NOT RESET;
DEF_Marche_Imposs.DELAY		 := 	T#0ms;
DEF_Marche_Imposs();

(* Défaut d'arrêt de la pompe primaire non autorisée en automatique*)
DEF_Arret_Imposs.CONDITION	:=	NOT MANUAL AND NOT CO_On AND STATE_ON
								AND( NOT EN_Off_INT OR NOT EN_Off_EXT)
								AND NOT RESET;
DEF_Arret_Imposs.DELAY		 := 	T#0ms;
DEF_Arret_Imposs();

(*défaut d'arrêt automatique de la pompe *)
DEF_Arret_Auto.CONDITION 	:=	(NOT WATER
								OR  NOT EN_On_INT
								OR NOT EN_On_EXT)
								AND  VAR_PSx AND NOT RESET;
DEF_Arret_Auto.DELAY		:=	T#0ms;
DEF_Arret_Auto();

(* Défaut amorçage de la pompe *)
Def_ON.CONDITION 		:= 	VAR_PSx AND NOT STATE_On AND NOT RESET;
Def_ON();

(* Défaut arrêt de la pompe *)
Def_OFF.CONDITION 		:= 	NOT VAR_PSx AND STATE_ON;
Def_OFF();

(* Défaut désamorçage *)
FD_PSxM.CLK 				:= 	STATE_On;
DEF_Desamorcage.DELAY 		:= 	INT_TO_TIME(0);
DEF_Desamorcage.CONDITION 	:= 	FD_PSxM.Q AND VAR_PSx;
DEF_Desamorcage();

(* Défaut interne pompe *)
IF VAR_Error_active THEN
	STATE_Erreur := 6;
ELSIF VAR_Overtemp_ctrl_fault THEN
	STATE_Erreur := 5;
ELSIF VAR_Overtemp_pump_fault THEN
	STATE_Erreur := 4;
ELSIF VAR_Overbalance_fault THEN
	STATE_Erreur := 3;
ELSIF VAR_Com_int_fault THEN
	STATE_Erreur := 2;
ELSIF VAR_Maint_required THEN
	STATE_Erreur := 1;
ELSE
	STATE_Erreur := 0;
END_IF
DEF_Interne.DELAY 		:= 	INT_TO_TIME(0);
DEF_Interne.CONDITION 	:= 	(STATE_Erreur > 0);
DEF_Interne.VAL1		:=	INT_TO_STRING(STATE_Erreur);
DEF_Interne();

STATE_NOK		:=	DEF_Arret_Imposs.DEF OR DEF_Marche_Imposs.DEF OR DEF_Arret_Auto.DEF
					OR DEF_On.DEF OR DEF_Off.DEF;

(* Reset des ordres *)
IF RCP_M_PSx AND M_ON THEN
	M_ON := FALSE;
END_IF

END_FUNCTION_BLOCK

// ---- POUs/Composant/POMPES/BLOCK_RS232_ONBOARD.TcPOU
FUNCTION_BLOCK BLOCK_RS232_ONBOARD
(* Communication RS232 - pour module On-Board Brooks *)
(*Gestion d'une seule pompe*)

(****************historique des versions*****************************)

(* Version 1-0 - HG - VERSION INIITIALE*)

(*************************************************************************)

VAR_INPUT
	CO_Regen:					BOOL;							(* Demande de mise en régénération de la pompe *)
	CO_Etat:					BOOL;							(* Commande 1 = Marche de la pompe 0 = Arret de la pompe *)
	CO_Forcage:					BOOL;							(* Permet de forcer sur une trame particuliere numero de trame dans ValeurForcageCptSend *)

	CONF_Forcage:				USINT;			(* Numero de la trame qui doit etre forcer avec le bool ForcageCptSend *)
	RESET:						BOOL;			(* Reset du driver*)
	OFF:						BOOL;			(* Désactivation du driver *)

	CO_ModeManu:				BOOL;			(* Passage en envoi manuel *)
	CO_EnvoiManu:				BOOL;			(* Commande d'envoi en mode manuel *)
	PRM_TrameManu:				STRING;			(* Contient la trame pour l'envoi manuel *)

	DEF_Port_com:				PRCDEF;			(* Defaut du port de communication rs232*)

	IN_COM			AT %I* :	PcComInData;	(*  ~ {LinkedWith:TIID^RS232^Entrées^Status;TIID^RS232^Entrées^Data1;TIID^RS232^Entrées^Data2;TIID^RS232^Entrées^Data3;TIID^RS232^Entrées^Data4;TIID^RS232^Entrées^Data5;TIID^RS232^Entrées^Data6;TIID^RS232^Entrées^Data7;TIID^RS232^Entrées^Data8;TIID^RS232^Entrées^Data9;TIID^RS232^Entrées^Data10;TIID^RS232^Entrées^Data11;TIID^RS232^Entrées^Data12;TIID^RS232^Entrées^Data13;TIID^RS232^Entrées^Data14;TIID^RS232^Entrées^Data15;TIID^RS232^Entrées^Data16;TIID^RS232^Entrées^Data17;TIID^RS232^Entrées^Data18;TIID^RS232^Entrées^Data19;TIID^RS232^Entrées^Data20;TIID^RS232^Entrées^Data21;TIID^RS232^Entrées^Data22;TIID^RS232^Entrées^Data23;TIID^RS232^Entrées^Data24;TIID^RS232^Entrées^Data25;TIID^RS232^Entrées^Data26;TIID^RS232^Entrées^Data27;TIID^RS232^Entrées^Data28;TIID^RS232^Entrées^Data29;TIID^RS232^Entrées^Data30;TIID^RS232^Entrées^Data31;TIID^RS232^Entrées^Data32;TIID^RS232^Entrées^Data33;TIID^RS232^Entrées^Data34;TIID^RS232^Entrées^Data35;TIID^RS232^Entrées^Data36;TIID^RS232^Entrées^Data37;TIID^RS232^Entrées^Data38;TIID^RS232^Entrées^Data39;TIID^RS232^Entrées^Data40;TIID^RS232^Entrées^Data41;TIID^RS232^Entrées^Data42;TIID^RS232^Entrées^Data43;TIID^RS232^Entrées^Data44;TIID^RS232^Entrées^Data45;TIID^RS232^Entrées^Data46;TIID^RS232^Entrées^Data47;TIID^RS232^Entrées^Data48;TIID^RS232^Entrées^Data49;TIID^RS232^Entrées^Data50;TIID^RS232^Entrées^Data51;TIID^RS232^Entrées^Data52;TIID^RS232^Entrées^Data53;TIID^RS232^Entrées^Data54;TIID^RS232^Entrées^Data55;TIID^RS232^Entrées^Data56;TIID^RS232^Entrées^Data57;TIID^RS232^Entrées^Data58;TIID^RS232^Entrées^Data59;TIID^RS232^Entrées^Data60;TIID^RS232^Entrées^Data61;TIID^RS232^Entrées^Data62;TIID^RS232^Entrées^Data63;TIID^RS232^Entrées^Data64} *)
END_VAR

VAR_INPUT PERSISTENT
	(*Entité*)
	IsComponent:		BOOL;			(*entité : composant*)
	IdXML:				STRING;			(*nom entité : identifiant pour recherche dans dico*)
	TagXML:				UINT;			(*nom entité : identifiant pour recherche dans dico*)
	IdParent:			STRING;			(*MNEMO de l'appelant*)
	MNEMO:				STRING;			(*MNEMO de l'entité*)
END_VAR

VAR_OUTPUT
	STATE_Temperature:			ARRAY[0..1] OF REAL;				(* Donne la température de chaque étage d'une pompe *)
	STATE_Regen:				BOOL;			(* Donne l'etat de la regen *)
	STATE_Pompe:				BOOL;			(* Donne l'etat du moteur de la cryo *)
	OUT_Com 		AT %Q* : 	PcComOutData;	(*  ~ {LinkedWith:TIID^RS232^Sorties^Data1;TIID^RS232^Sorties^Data2;TIID^RS232^Sorties^Data3;TIID^RS232^Sorties^Data4;TIID^RS232^Sorties^Data5;TIID^RS232^Sorties^Data6;TIID^RS232^Sorties^Data7;TIID^RS232^Sorties^Data8;TIID^RS232^Sorties^Data9;TIID^RS232^Sorties^Data10;TIID^RS232^Sorties^Data11;TIID^RS232^Sorties^Data12;TIID^RS232^Sorties^Data13;TIID^RS232^Sorties^Data14;TIID^RS232^Sorties^Data15;TIID^RS232^Sorties^Data16;TIID^RS232^Sorties^Data17;TIID^RS232^Sorties^Data18;TIID^RS232^Sorties^Data19;TIID^RS232^Sorties^Data20;TIID^RS232^Sorties^Data21;TIID^RS232^Sorties^Data22;TIID^RS232^Sorties^Data23;TIID^RS232^Sorties^Data24;TIID^RS232^Sorties^Data25;TIID^RS232^Sorties^Data26;TIID^RS232^Sorties^Data27;TIID^RS232^Sorties^Data28;TIID^RS232^Sorties^Data29;TIID^RS232^Sorties^Data30;TIID^RS232^Sorties^Data31;TIID^RS232^Sorties^Data32;TIID^RS232^Sorties^Data33;TIID^RS232^Sorties^Data34;TIID^RS232^Sorties^Data35;TIID^RS232^Sorties^Data36;TIID^RS232^Sorties^Data37;TIID^RS232^Sorties^Data38;TIID^RS232^Sorties^Data39;TIID^RS232^Sorties^Data40;TIID^RS232^Sorties^Data41;TIID^RS232^Sorties^Data42;TIID^RS232^Sorties^Data43;TIID^RS232^Sorties^Data44;TIID^RS232^Sorties^Data45;TIID^RS232^Sorties^Data46;TIID^RS232^Sorties^Data47;TIID^RS232^Sorties^Data48;TIID^RS232^Sorties^Data49;TIID^RS232^Sorties^Data50;TIID^RS232^Sorties^Data51;TIID^RS232^Sorties^Data52;TIID^RS232^Sorties^Data53;TIID^RS232^Sorties^Data54;TIID^RS232^Sorties^Data55;TIID^RS232^Sorties^Data56;TIID^RS232^Sorties^Data57;TIID^RS232^Sorties^Data58;TIID^RS232^Sorties^Data59;TIID^RS232^Sorties^Data60;TIID^RS232^Sorties^Data61;TIID^RS232^Sorties^Data62;TIID^RS232^Sorties^Data63;TIID^RS232^Sorties^Data64} *)
	(*OUT_DTR_RTS 	AT %Q* : 		UINT;*)
	STATE_Ready:				BOOL;			(* Driver en fonctionnement *)
	STATE_NOK:					BOOL;			(* Driver en défaut *)
END_VAR

VAR
	TIMER_Cadence: 				TON;			(*Timer cadencement communication*)
	TIMER_Demarrage: 			TON;
	VAR_Cadence:				USINT;			(*Numéro de la trame en cours*)
	VAR_Mem_Cadence:			USINT;			(*Mémorisation numéro dela trame*)

	OUT_Send_Data:				SendString;		(*Fonction d'envoi*)
	OUT_Buffer: 				ComBuffer;		(*Buffer trame d'envoi *)

	IN_Receive_Data:			ReceiveString;	(*Fonction de réception*)
	IN_Buffer: 					ComBuffer;		(*Buffer trame de réception *)

	VAR_ClearBuffer: 			ClearComBuffer;	(*Fonction de RAZ buffer*)

	(* background communication with the COM port device *)
	VAR_COMportControl: 		SerialLineControl;
	VAR_COMportControlError: 	BOOL;
	VAR_COMportControlErrorID: 	ComError_t;

	VAR_NB:						USINT;
	VAR_NB2:					USINT;
	VAR_BuffString:				STRING;
	VAR_TrameRetour:			STRING;
	VAR_STR1:					STRING[1];
	VAR_STR2:					STRING[1];
	VAR_ReceptionOk:			BOOL;

	FM_On:						R_TRIG;
	FM_Off:						F_TRIG;
	FM_Regen:					R_TRIG;
	VAR_Mem_CO_On:				BOOL;
	VAR_Mem_CO_Off:				BOOL;
	VAR_Mem_CO_Regen:			BOOL;
END_VAR

(*Cadence :
Trame 1 : Demande état marche/arrêt - A?
Trame 2 : Demande état regen - O
Trame 3: Demande température étage 1 - J
Trame 4 : Demande température étage 2 - K
Trame 5 : Demande de marche ou d'arrêt d'une pompe - A1 / A0
Trame 6:  Demande de regen d'une pompe - N1 / N0
*)

(* Paramètre statique *)
IdXML							:=	'8';
TagXML							:=	2;

DEF_Port_com.IdXml				:=	'11';
DEF_Port_com.TagXml				:=	1;

(*Gestion des fronts demandes*)
FM_On.CLK	:=	CO_Etat;
FM_On();
IF FM_On.Q THEN
	VAR_Mem_CO_On	:=	TRUE;
END_IF
FM_Off.CLK	:=	CO_Etat;
FM_Off();
IF FM_Off.Q THEN
	VAR_Mem_CO_Off	:=	TRUE;
END_IF
FM_Regen.CLK	:=	CO_Regen;
FM_Regen();
IF FM_Regen.Q THEN
	VAR_Mem_CO_Regen	:=	TRUE;
END_IF

(*RESET ou DESACTIVATION Driver*)
IF RESET OR OFF THEN
	STATE_Temperature[0]	:=	0;
	STATE_Temperature[1]	:=	0;
	VAR_Mem_CO_On		:=	FALSE;
	VAR_Mem_CO_Off		:=	TRUE;
	VAR_Mem_CO_Regen		:=	FALSE;
	RETURN;
END_IF

TIMER_Demarrage.IN 	:= 	NOT IN_Receive_Data.Busy AND NOT OUT_Send_Data.Busy AND NOT VAR_ReceptionOk;
TIMER_Demarrage.PT	:=	T#5s;
TIMER_Demarrage();
IF TIMER_Demarrage.Q  THEN
	VAR_ReceptionOk	:=	TRUE;
	VAR_Cadence 		:= 	1;
END_IF

(*Cadencement des trames*)
TIMER_Cadence(IN:=VAR_ReceptionOk, PT:=T#500ms);
VAR_Mem_Cadence	:=	VAR_Cadence;

(*GESTION ENVOI*)
IF TIMER_Cadence.Q AND NOT OUT_Send_Data.Busy AND NOT CO_ModeManu THEN
	VAR_STR2 := CHR(36);	(*$ = hex 24 = dec 36*)

	(* Remplissage trame : $ + code + checksum + 0D*)
	CASE VAR_Cadence OF

			1: 	(* Demande état on/off pompe*)
				VAR_BuffString		:= 	'';
				VAR_BuffString		:=	VAR_STR2;
				VAR_BuffString		:=	CONCAT(VAR_BuffString, 'A?');
				VAR_BuffString		:=	CONCAT(VAR_BuffString,CHECKSUM(VAR_BuffString,TRUE));
				VAR_BuffString		:=	CONCAT(VAR_BuffString,'$0D');
				OUT_Send_Data.SendString		:=	VAR_BuffString;

			2: 	(* Demande état regen pompe*)
				VAR_BuffString		:= 	'';
				VAR_BuffString		:=	VAR_STR2;
				VAR_BuffString		:=	CONCAT(VAR_BuffString, 'O');
				VAR_BuffString		:=	CONCAT(VAR_BuffString,CHECKSUM(VAR_BuffString,TRUE));
				VAR_BuffString		:=	CONCAT(VAR_BuffString,'$0D');
				OUT_Send_Data.SendString		:=	VAR_BuffString;

			3: 	(* Demande température étage 1*)
				VAR_BuffString		:= 	'';
				VAR_BuffString		:=	VAR_STR2;
				VAR_BuffString		:=	CONCAT(VAR_BuffString, 'J');
				VAR_BuffString		:=	CONCAT(VAR_BuffString,CHECKSUM(VAR_BuffString,TRUE));
				VAR_BuffString		:=	CONCAT(VAR_BuffString,'$0D');
				OUT_Send_Data.SendString		:=	VAR_BuffString;

			4: 	(* Demande température étage 2*)
				VAR_BuffString		:= 	'';
				VAR_BuffString		:=	VAR_STR2;
				VAR_BuffString		:=	CONCAT(VAR_BuffString, 'K');
				VAR_BuffString		:=	CONCAT(VAR_BuffString,CHECKSUM(VAR_BuffString,TRUE));
				VAR_BuffString		:=	CONCAT(VAR_BuffString,'$0D');
				OUT_Send_Data.SendString		:=	VAR_BuffString;

			5: 	(* Demande de marche ou d'arrêt d'une pompe *)
				VAR_BuffString		:= 	'';
				VAR_BuffString		:=	VAR_STR2;
				IF	CO_ETAT THEN
					VAR_BuffString	:=	CONCAT(VAR_BuffString,'A1');
				ELSE
					VAR_BuffString	:=	CONCAT(VAR_BuffString,'A0');
				END_IF
				VAR_BuffString		:=	CONCAT(VAR_BuffString,CHECKSUM(VAR_BuffString,TRUE));
				VAR_BuffString		:=	CONCAT(VAR_BuffString,'$0D');
				OUT_Send_Data.SendString		:=	VAR_BuffString;

			6:	(* Demande de regen d'une pompe *)
				VAR_BuffString		:= 	'';
				VAR_BuffString		:=	VAR_STR2;
				VAR_BuffString		:=	CONCAT(VAR_BuffString,'N1');
				VAR_BuffString		:=	CONCAT(VAR_BuffString,CHECKSUM(VAR_BuffString,TRUE));
				VAR_BuffString		:=	CONCAT(VAR_BuffString,'$0D');
				OUT_Send_Data.SendString		:=	VAR_BuffString;
	END_CASE

	(*Envoi*)
	OUT_Send_Data(TXbuffer:= OUT_Buffer);

	(* Reset timer *)
	VAR_ReceptionOk := FALSE;
ELSE
	IF CO_ModeManu AND CO_EnvoiManu THEN
		OUT_Send_Data.SendString	:=	VAR_BuffString;
		(*Envoi*)
		OUT_Send_Data(TXbuffer:= OUT_Buffer);
		CO_EnvoiManu		:=	FALSE;
		VAR_ReceptionOk 	:= 	FALSE;
	END_IF
END_IF

IF CO_ModeManu THEN
		VAR_STR1 		:= 	CHECKSUM(PRM_TrameManu ,FALSE);
		VAR_STR2		:=	CHR(36);
		VAR_BuffString	:=	CONCAT(VAR_STR2,PRM_TrameManu);
		VAR_BuffString	:=	CONCAT(VAR_BuffString,VAR_STR1);
		VAR_BuffString	:=	CONCAT(VAR_BuffString,CHR(13));
END_IF

(*GESTION RECEPTION*)
(*Réception*)
IN_Receive_Data(
	(*Prefix := '$',*)
	Suffix:= '$0D',
	Timeout:= T#1s,
	Reset :=OFF,
	ReceivedString := VAR_TrameRetour,
	RXbuffer := IN_Buffer);

(*interprétation trame retour*)
IF IN_Receive_Data.StringReceived THEN
	IF NOT CO_ModeManu THEN
		CASE VAR_Cadence OF

			1: (* Demande état On/off pompe *)
				VAR_STR1	:=	MID(VAR_TrameRetour,1,3);
				STATE_Pompe	:=	(VAR_STR1 = '1');

			2: (* Demande état regen pompe *)
				VAR_STR1	:=	MID(VAR_TrameRetour,1,3);
				STATE_Regen	:=	NOT((VAR_STR1 = 'V') OR (VAR_STR1 = 'P'));

			3: (* demande température étage 1*)
				STATE_Temperature[0]	:=	STRING_TO_REAL(MID(VAR_TrameRetour,6,4));

			4: (* demande température étage 2*)
				STATE_Temperature[1]	:=	STRING_TO_REAL(MID(VAR_TrameRetour,6,4));

			5: (* Demande de marche ou d'arrêt d'une pompe *)
				VAR_Mem_CO_Off	:=	FALSE;
				VAR_Mem_CO_On	:=	FALSE;

			6: (* Demande de regen d'une pompe *)
				CO_REGEN			:=	FALSE;
				VAR_Mem_CO_Regen	:=	FALSE;
		END_CASE

		(*trame suivante*)
		IF NOT CO_Forcage THEN
			IF VAR_Mem_CO_Regen THEN
				VAR_Cadence := 6;
			ELSIF VAR_Mem_CO_Off OR VAR_Mem_CO_On THEN
				VAR_Cadence := 5;
			ELSE
				VAR_Cadence := VAR_Cadence + 1;
				IF VAR_Cadence >= 5 THEN
					VAR_Cadence	:=	1;
				END_IF
			END_IF
		ELSE
			VAR_Cadence 	 := 	CONF_Forcage;
		END_IF
	END_IF

	VAR_ReceptionOk := TRUE;

	(*Effacement buffer réception*)
	VAR_ClearBuffer(Buffer := IN_Buffer);
END_IF

(* GESTION COMMUNICATION *)
VAR_COMportControl(
	Mode:= SERIALLINEMODE_PC_COM_PORT,
	pComIn:= ADR(IN_COM),
	pComOut:= ADR(OUT_COM),
	SizeComIn:=SIZEOF(IN_COM),
	TxBuffer:= OUT_Buffer,
	RxBuffer:= IN_Buffer,
	Error=> VAR_COMportControlError,
	ErrorID=> VAR_COMportControlErrorID );

(*GESTION DEFAUTS*)
Def_port_com.DELAY :=T#0s;
Def_port_com.CONDITION := VAR_COMportControlError;
Def_port_com();

(*Etat*)
STATE_Ready		:=	NOT OFF;
STATE_NOK			:=	Def_port_com.DEF;

END_FUNCTION_BLOCK

// ---- POUs/Composant/SERVITUDES/BLOCK_CHILLER.TcPOU
FUNCTION_BLOCK BLOCK_CHILLER

(* Gestion d'un groupe de circulation d'eau froide, avec retour de défaut, et commande de mise en marche (pas de controle de marche)*)

(****************historique des versions*****************************)

(* Version 1-0 - AB : affaire 7506*)

(*************************************************************************)

VAR_INPUT
	I_PARAM_SYSTEM_OK:	BOOL;														(*paramétrage système ok*)
	MANUAL:				BOOL;				(* ~ (OPC : 1 : available for OPC-clients) *)		(* Mode de pilotage manuel *)
	RESET:				BOOL;														(* Condition de réiinitialisation de la fonction *)

	DEF_Chill:			PRCDEF;			(*Défaut de groupe froid*)

	CO_On:				BOOL;			(*demande de marche en mode automatique généré par la fonction qui gère la pompe*)

	IN_Def:				BOOL;		(*Groupe en defaut*)
	OUT_On:				BOOL;		(* Marche groupe *)

END_VAR

VAR_INPUT PERSISTENT
	CONF_Tim_Valid_On:			TIME:=T#0ms;	(*temporisation de validation du l'état STATE_OK*)
	CONF_Tim_Valid_Off:			TIME:=T#0ms;	(*temporisation de validation de l'état STATE_AR*)

	(*Entité*)
	IsComponent:		BOOL;			(*entité : composant*)
	IdXML:				STRING;			(*nom entité : identifiant pour recherche dans dico*)
	TagXML:				UINT;			(*nom entité : identifiant pour recherche dans dico*)
	IdParent:			STRING;			(*MNEMO de l'appelant*)
	MNEMO:				STRING;			(*MNEMO de l'entité*)
END_VAR

VAR_OUTPUT
	(*variable d'état d'autorisation*)
	AUTOR_On_IHM:				BOOL;			(* ~ (OPC : 1 : available for OPC-clients) *)	(*indique que la mise en marche de la pompe est autorisée en mode manuel depuis l'IHM*)
	AUTOR_Off_IHM:				BOOL;			(* ~ (OPC : 1 : available for OPC-clients) *)	(*indique que l'arrêt de la pompe est autorisée en mode manuel depuis l'IHM*)

	STATE_On:					BOOL;			(* ~ (OPC : 1 : available for OPC-clients) *)	(*indique que la pompe est en marche et à atteint sa vitesse*)
	STATE_NOK:					BOOL;			(* ~ (OPC : 1 : available for OPC-clients) *)	(*indique la présence d'un défaut sur la pompe ou que l'ordre de marche a été refusé*)
	STATE_Off:					BOOL;			(* ~ (OPC : 1 : available for OPC-clients) *)	(*indique que la pompe est à l'arrêt*)
END_VAR

VAR
	TIMER_Valid_On:				TON;
	TIMER_Valid_Off:			TON;
	(* Variables pour les sorties profibus *)

	(* Variables demande en mode manuel*)
	M_On:						BOOL;					(* ~ (OPC : 1 : available for OPC-clients) *)	(* Ordre marche/arrêt de la  pompe en mode manuel *)
	RCP_M_On:					BOOL;														(* bit de reception de l'ordre de marche en mode manuel*)
	VAR_On:						BOOL;														(* variable intermédiaire de marche de la pompe*)

	VAR_CPT:					BLOCK_CPT_TEMPS;
END_VAR

IdXML						:=	'10';
TagXML						:=	2;

(*Défaut interne*)
DEF_Chill.IdXML				:=	'0';
DEF_Chill.TagXML			:=	6;

(* Gestion des ordres en mode manuel *)
RCP_M_On 					:=	M_On;

(*gestion des bits d'autorisation en mode manuel*)
AUTOR_On_IHM			:=	NOT RESET AND NOT VAR_On  AND MANUAL;
AUTOR_Off_IHM			:=	NOT RESET  AND VAR_On  AND MANUAL;

(* Défaut du groupe froid*)
DEF_Chill.CONDITION		:=		IN_Def;
DEF_Chill.DELAY			:=		T#1s;
DEF_Chill();


(* ARRET groupe*)
IF 		(NOT CO_On AND NOT MANUAL)
		OR ( RCP_M_On AND AUTOR_Off_IHM) OR RESET
		THEN
			Var_On 				:= 	FALSE;
(*MARCHE POMPES*)
ELSIF	( CO_On AND NOT MANUAL)
		 OR 	( RCP_M_On AND AUTOR_On_IHM) THEN
			Var_On 				:= 	TRUE;
END_IF;

(*SORTIE MARCHE GROUPE*)
OUT_On			:= 	VAR_On;


(*affectation des bits d'état*)
(*indicateur pompe en marche STATE_ON*)
TIMER_Valid_On.IN	:=	OUT_On;
TIMER_Valid_On(PT:=CONF_Tim_Valid_On);
STATE_ON			:=	TIMER_Valid_On.Q;
(*indicateur pompe à l'arrêt STATE_OFF*)
TIMER_Valid_Off.IN	:=	NOT OUT_On;
TIMER_Valid_Off(PT:=CONF_Tim_Valid_Off);
STATE_Off			:=	TIMER_Valid_Off.Q;

STATE_NOK			:=	DEF_Chill.DEF;


(*Gestion compteur*)
VAR_CPT(I_On:= STATE_On);


(* Reset des ordres*)
IF M_On AND RCP_M_On THEN
	M_On		:= FALSE;
END_IF;

END_FUNCTION_BLOCK

// ---- POUs/Composant/SERVITUDES/BLOCK_CTA_HOT_COLD.TcPOU
FUNCTION_BLOCK BLOCK_CTA_HOT_COLD

(* Gestion d'un groupe de circulateur eau chaude/eau froide *)

VAR_INPUT
	I_PARAM_SYSTEM_OK:	BOOL;																	(*paramétrage système ok*)
	MANUAL:				BOOL;				(* ~ (OPC : 1 : available for OPC-clients) *)		(* Mode de pilotage manuel *)
	RESET:				BOOL;																	(* Condition de réiinitialisation de la fonction *)


	CO_Froid:			BOOL;	(*demande de marche en mode automatique eau froide*)
	CO_Chaud:			BOOL;	(*Demande de marche en mode automatique groupe chaud*)

	PRM_Temperature:	BOOL;	(*Consgine de temperature eau chaude, 0 = 40°C, 1 = 80°C*)


END_VAR

VAR_INPUT PERSISTENT
	CONF_Tim_Valid_On:		TIME:=T#0MS;	(*temporisation de validation du l'état STATE_OK*)
	CONF_Tim_Valid_Off:		TIME:=T#0MS;	(*temporisation de validation de l'état STATE_AR*)

	(*Entité*)
	IsComponent:		BOOL;			(*entité : composant*)
	IdXML:				STRING;			(*nom entité : identifiant pour recherche dans dico*)
	TagXML:				UINT;			(*nom entité : identifiant pour recherche dans dico*)
	IdParent:			STRING;			(*MNEMO de l'appelant*)
	MNEMO:				STRING;			(*MNEMO de l'entité*)
END_VAR
VAR_OUTPUT
	OUT_Chaud:				BOOL;		(*Marche groupe chaud*)
	OUT_Froid:				BOOL;		(*Marche groupe froid*)

	AUTOR_On_IHM:			BOOL;			(* ~ (OPC : 1 : available for OPC-clients) *)	(*indique que la mise en marche de la pompe est autorisée en mode manuel depuis l'IHM*)
	AUTOR_Off_IHM:			BOOL;			(* ~ (OPC : 1 : available for OPC-clients) *)	(*indique que l'arrêt de la pompe est autorisée en mode manuel depuis l'IHM*)

	STATE_On:				BOOL;			(* ~ (OPC : 1 : available for OPC-clients) *)	(*indique que la pompe est en marche et à atteint sa vitesse*)
	STATE_NOK:				BOOL;			(* ~ (OPC : 1 : available for OPC-clients) *)	(*indique la présence d'un défaut sur la pompe ou que l'ordre de marche a été refusé*)
	STATE_Off:				BOOL;			(* ~ (OPC : 1 : available for OPC-clients) *)	(*indique que la pompe est à l'arrêt*)

	AO_CTA_SET:			ANALOG_OUTPUT;
	OUT_CTA_SET:		INT;			(*Sortie consigne temperature eau chaude*)

END_VAR
VAR

	(*Variable de demande marche en mode manuel*)
	M_On_HOT:					BOOL;	(* ~ (OPC : 1 : available for OPC-clients) *)	(* Ordre marche/arrêt eau chaude *)
	M_On_COLD:					BOOL;	(* ~ (OPC : 1 : available for OPC-clients) *)	(* Ordre marche/arrêt eau froide *)

	RCP_M_On_HOT:				BOOL;	(* bit de reception de l'ordre de marche eau chaude en mode manuel*)
	RCP_M_On_COLD:				BOOL;	(* bit de reception de l'ordre de marche eau froide en mode manuel*)

	TIMER_Valid_On_HOT:			TON;
	TIMER_Valid_Off_HOT:		TON;
	TIMER_Valid_COLD:			TON;
	TIMER_Valid_Off_COLD:		TON;


	VAR_On_HOT:					BOOL;			(*Variable intermediaire de marche eau chaude*)
	VAR_On_COLD:				BOOL;			(*Variable intermediaire de marche eau froide*)

	(* Variables pour les sorties profibus *)

	VAR_CPT:					BLOCK_CPT_TEMPS;
END_VAR

IdXML							:=	'10';
TagXML							:=	2;

END_FUNCTION_BLOCK

// ---- POUs/Composant/SERVITUDES/BLOCK_SV4200.TcPOU
FUNCTION_BLOCK BLOCK_SV4200
//  Fonction de gestion d'un débitmètre avec retour température et débit

//HISTORIQUE				
//VERSION 0.0 - 06/2023 - GV - (Basé sur version la version 3.0 du block d'Hélène des HC)
					//Adaptation pour machine de dépôt
					//Modification pour gestion AC4000 avec Struct_IHM 

VAR_INPUT
	RESET:					BOOL;			(*entrée de reset de la fonction*)

	I_Device_OK:			BOOL;			(*INPUT carte OP - données exploitables*)
	IN_ProcessData0	AT %I*:	USINT;			(*INPUT IO-link Data process*)
	IN_ProcessData1	AT %I*:	USINT;			(*INPUT IO-link Data process*)
	IN_ProcessData2	AT %I*:	USINT;			(*INPUT IO-link Data process*)
	IN_ProcessData3	AT %I*:	USINT;			(*INPUT IO-link Data process*)
	IN_ChannelState AT %I*:	USINT;			(*INPUT Device Channel State*)
	
	DEF_Channel:			PRCDEF;			(*défaut channel IO-link*)
	DEF_Flow:				PRCDEF;			(*défaut débit hors limites*)
	DEF_Temp:				PRCDEF;			(*défaut température hors limites*)	
	
	(*ELEMENTS DE CONFIGURATION*)
	(*Entité*)
	IsComponent:			BOOL;			(*entité : assemblage*)
	IdXML:					STRING;			(*nom entité : identifiant pour recherche dans dico*)
	TagXML:					UINT;			(*nom entité : identifiant pour recherche dans dico*)
	IdParent:				STRING;			(*MNEMO de l'appelant*)
	MNEMO:					STRING;			(*MNEMO de l'entité*)	
END_VAR

VAR_OUTPUT
	STATE_OK:				BOOL;			(* O_STANDARD -- entité fonctionnelle*)
	STATE_NOK:				BOOL;			(* O_STANDARD -- entité en défaut - pour affichage*)
	STATE_Flow:				REAL;			(*débit courant en l/s*)
	STATE_Temp:				REAL;			(*température courante en °C*)
END_VAR

VAR
	VAR_Valid_Elmt:			BOOL;
	VAR_W_Calcul1:			WORD;
	VAR_W_Calcul2:			WORD;
	VAR_W_Calcul3:			WORD;
	VAR_Int_Calcul:			INT;
END_VAR

VAR_EXTERNAL
END_VAR

IdXML					:=	'10';
TagXML					:=	5;

(*TAG DEFAUTS*)
DEF_Channel.IdXML		:=	'8';
DEF_Channel.TagXML		:=	12;
DEF_Flow.IdXML			:=	'8';
DEF_Flow.TagXML			:=	13;
DEF_Temp.IdXML			:=	'8';
DEF_Temp.TagXML			:=	14;

(*MESURE VALIDE*)
(*Défaut channel IO-link - CTRLOK*)
DEF_Channel.CONDITION		:=	NOT RESET AND I_Device_OK AND (IN_ChannelState<>3);
DEF_Channel.DELAY			:=	T#1S;
DEF_Channel.VAL1			:=	USINT_TO_STRING(IN_ChannelState);
DEF_Channel();
VAR_Valid_Elmt				:=	NOT RESET AND I_Device_OK AND NOT DEF_Channel.DEF;
	
(*DEBIT - PVD2 dans la doc - correspondant à octet 0 et octet 1*)
VAR_W_Calcul1	:= ROL(BYTE_TO_WORD(IN_ProcessData0),8); (*décalage de l'octet*)
VAR_W_Calcul2	:= BYTE_TO_WORD(IN_ProcessData1);
VAR_W_Calcul3	:= VAR_W_Calcul1 OR VAR_W_Calcul2; (*concaténation des 2 octets*)
VAR_Int_Calcul 	:=	WORD_TO_INT(VAR_W_Calcul3);
STATE_Flow		:=	INT_TO_REAL(VAR_Int_Calcul)/10.0;
(*Défaut débit hors limite : 260 - CTRLOK*)
DEF_Flow.CONDITION		:=	VAR_Valid_Elmt AND (VAR_Int_Calcul > 260);
DEF_Flow.DELAY			:=	T#1S;
DEF_Flow();

(*TEMPERATURE - PVD1 dans la doc moins les 2 premiers bits - correspondant à octet 2 et octet 3*)
VAR_W_Calcul1	:= ROL(BYTE_TO_WORD(IN_ProcessData2),8); (*décalage de l'octet*)
VAR_W_Calcul2	:= BYTE_TO_WORD(IN_ProcessData3);
VAR_W_Calcul3	:= SHR(VAR_W_Calcul1 OR VAR_W_Calcul2,2); (*concaténation des 2 octets et décalage de 2 bits pour supprimer*)
VAR_Int_Calcul 	:=	WORD_TO_INT(VAR_W_Calcul3);
STATE_Temp		:=	INT_TO_REAL(VAR_Int_Calcul)/10.0;
(*Défaut temperature hors limite : 1105 / -305 - CTRLOK*)
DEF_Temp.CONDITION		:=	VAR_Valid_Elmt AND ((VAR_Int_Calcul>1105) OR (VAR_Int_Calcul<-305));
DEF_Temp.DELAY			:=	T#1S;
DEF_Temp();


(*ETATS GENERAUX*)
STATE_OK		:=	VAR_Valid_Elmt AND NOT DEF_Flow.DEF AND NOT DEF_Temp.DEF;
STATE_NOK		:=	NOT RESET AND (DEF_Channel.DEF OR DEF_Flow.DEF OR DEF_Temp.DEF);

END_FUNCTION_BLOCK

// ---- POUs/Composant/VANNES/BLOCK_VVAT_650_ETHERCAT.TcPOU
FUNCTION_BLOCK BLOCK_VVAT_650_ETHERCAT

(* Gestion d'une vanne 3 positions VAT interface ethercat*)

(****************historique des versions*****************************)

(* Version 1-0 - AB - VERSION INITIALE AC2000 - aff 9015 *)
(* Version 2-0 - GV - 06-2015 - affaire 9070 - Adaptation pour journal des évènements externe*)

(*
Configuration vanne : Startup CoE :
Param 0x20F5 _ valeur 0x02 ==> sensor 1 unit à mbar

Configuration vanne via le logiciel VAT CPA , dans terminal :
envoi de la commande 		a:74031 
Cette commande sert à mettre la réception de la pression jauge sur external digital output sensor 1

envoi de la commande			s:2309000000
Cette commande sert à mettre le signal de reception jauge sur un DINT, range par défaut ==> sans doute inutile de la mettre	

Signal de la jauge process envoyée au bloc par entrée I_Pressure (REAL)
Information pression envoyée à la vanne par OUT_Pression_Ethercat (DINT, avec max range de 1 000 000)

*)


(*************************************************************************)


VAR_INPUT
(*paramètre standard*)
	RESET:   					BOOL; 											(*Condition RAZ actionneur*)
	MANUAL:  					BOOL; 	(* ~ (OPC : 1 : available for OPC-clients) *)		(*Mode manuel*)

(*entrée externe*)
	IN_OFF:						BOOL; 	(* ~ (OPC : 1 : available for OPC-clients) *)		(*E.TOR vanne fermée*)
	IN_ON:						BOOL; 	(* ~ (OPC : 1 : available for OPC-clients) *)		(*E.TOR vanne ouverte*)

	IN_POSITION		AT%I*:		DINT;	(*Retour de position de la jauge, de 0 à 100 000 points*)
	I_PRESSION:					REAL;	(*Mesure de pression externe*)

(*Paramètres*)
	PRM_Mode:					BOOL; 	(* ~ (OPC : 1 : available for OPC-clients) *)		(*Mode FALSE = Position / TRUE = Pression*)
	PRM_Pression:				REAL; 	(* ~ (OPC : 1 : available for OPC-clients) *)		(*Consigne de pression - en unité cohérente avec la mesure*)
	PRM_Position:				REAL;	(* ~ (OPC : 1 : available for OPC-clients) *)		(*Consigne de position de la vanne en %*)
	PRM_W_Pr_HI:				REAL;	(* ~ (OPC : 1 : available for OPC-clients) *)		(*Tolérance haute de stabilisation de pression pour obtention de l'état stab pression ok*)
	PRM_W_Pr_LO:				REAL;	(* ~ (OPC : 1 : available for OPC-clients) *)		(*Tolérance basse de dtabilisation de pression pour obtention de l'état stab pression ok*)
	PRM_Tim_W_Pr:				TIME;	(* ~ (OPC : 1 : available for OPC-clients) *)		(*Temps de validation de stabilisation de la pression*)

(*défaut du bloc*)
	DEF_On:  					PRCDEF; 										(*00 - Défaut d'ouverture de la vanne*)
	DEF_Off:   					PRCDEF; 										(*01 - Défaut de fermeture de la vanne*)
	DEF_On_Imposs:				PRCDEF;										(*03 - Défaut d'ouverture ou de mise en laminage non autorisée en mode automatique*)
	DEF_Off_Imposs:				PRCDEF;										(*04 - Défaut de fermeture non autorisée en mode automatique*)
	DEF_Off_auto:				PRCDEF;										(*05 - Défaut de fermeture automatique de la vanne*)
	DEF_Position:				PRCDEF;										(*06 - Défaut d'obtention de la position*)
	DEF_Pression:				PRCDEF;										(*07 - Défaut d'obtention de la pression*)
	DEF_Surv_Pression:			PRCDEF;										(*08 - Défaut de surveillance de la pression - perte du critère de stabilisation*)
	ALA_Surv_Pression:			PRCDEF;										(*09 - Alarme de surveillance de la rpession - perte du critère de stabilisation*)

(*parametre de pilotage en entrée*)
	CO_On:   					BOOL; 											(*Ordre mode automatique ouverture*)
	CO_Lam:						BOOL;											(*Ordre mode automatique laminage*)
	EN_On_INT:   				BOOL;											(*Condition d'autorisation d'ouverture ou de laminage donnée par le bloc qui instancie le bloc actuator*)
	EN_Off_INT:  				BOOL; 											(*Condition d'autorisation de fermeture donnée par le bloc qui instacie le bloc actuator*)
	EN_On_EXT:					BOOL:=TRUE;									(*condition d'autorisation d'ouverture ou de laminage externe*)
	EN_Off_EXT:					BOOL:=TRUE;									(*condition d'autorisation de fermeture externe*)
END_VAR

VAR_INPUT PERSISTENT
(*parametre de configuration constructeur*)
(*les parametres suivants dépendent de la configuration de la machine*)
	CONF_Tim_Valid_On:  		TIME:=T#100MS; 			(*Temps validation de la position ouverte *)
	CONF_Tim_Valid_Off:   		TIME:=T#100ms; 			(*Temps validation de la position fermée *)
	CONF_EN_On:					USINT:=0;				(*définit la réaction du système en cas de perte des conditions d'autorisation d'activation EN_On*)
														(* 0 = désactivation automatique  en cas de perte des conditions d'autorisation d'activation uniquement en manuel*)
														(* 1 = désactivation automatique en cas de perte des conditions d'autorisation d'activation en auto et en manuel*)
														(* 2 = Pas de déscativation automatique*)
	CONF_Pr_Max_SP:			REAL;					(* Consigne max. de pression en pleine echelle 10V - correspond à la pleine échelle du capteur connecté au coffret*)
	CONF_WPos:				REAL;					(*Tolérance de positionnement pour obtention de l'état STATE_POS_ok*)
	CONF_Tim_WPos:			TIME;					(*Temps de validation de l'état STATE_POS_Ok*)
	PRM_Max_Tim_W:			TIME;	(* ~ (OPC : 1 : available for OPC-clients) *)		(*Temps Max d'obtention de l'état stabilisation pression ok*)
	PRM_Tim_Def_Pr:			TIME;	(* ~ (OPC : 1 : available for OPC-clients) *)		(*Temps d'enveloppe du défaut de surveillance de la pression*)
	PRM_Tim_Ala_Pr:			TIME;	(* ~ (OPC : 1 : available for OPC-clients) *)		(*Temps d'enveloppe de l'alarme de surveillance de la pression*)

	(*Entité*)
	IsComponent:	BOOL;			(*entité : composant*)
	IdXML:			STRING;			(*nom entité : identifiant pour recherche dans dico*)
	TagXML:			UINT;			(*nom entité : identifiant pour recherche dans dico*)
	IdParent:		STRING;			(*MNEMO de l'appelant*)
	MNEMO:			STRING;			(*MNEMO de l'entité*)
END_VAR

VAR_OUTPUT
	OUT_Pressure				AT%Q*:	DINT;	(*envoi de la pression reçue par jauge sur trame ethercat, codée sur 1 000 000 point pour pleine échelle*)
	OUT_Control_Mode			AT%Q*:	USINT;	(*control mode : 2-position, 3-close, 4-open, 5-pression*)
	OUT_Pressure_Setpoint		AT%Q*:	DINT;	(*consigne puissance, codé sur 1 000 000 points pour pleine echelle*)
	OUT_Position_Setpoint		AT%Q*:	DINT;	(*consigne position , codé sur 100 000 point pour 100%*)

	STATE_On:	   				BOOL; 	(* ~ (OPC : 1 : available for OPC-clients) *)		(*Indicateur ouverture ok*)
	STATE_Off:  				BOOL; 	(* ~ (OPC : 1 : available for OPC-clients) *)		(*Indicateur fermeture ok*)
	STATE_Nok:					BOOL;	(* ~ (OPC : 1 : available for OPC-clients) *)		(*Indicateur défaut sur la vanne*)
	STATE_Lam:					BOOL;	(* ~ (OPC : 1 : available for OPC-clients) *)		(*Indicateur mise en laminage ok *)
	STATE_Pos_Ok:				BOOL;	(* ~ (OPC : 1 : available for OPC-clients) *)		(*Indicateur de positionnement de la vanne ok *)
	STATE_Press_Ok:				BOOL;	(* ~ (OPC : 1 : available for OPC-clients) *)		(*Indicateur de stabilisation de la pression ok *)
	STATE_Ok:					BOOL;	(* ~ (OPC : 1 : available for OPC-clients) *)		(*Indicateur de stabilisation autour du point de consigne de pression
																				ou de positionnement ok si le controle est en mode position*)
	STATE_Position:				REAL;	(* ~ (OPC : 1 : available for OPC-clients) *)		(*Retour de position de la vanne*)
	STATE_Setpoint:				REAL;	(* ~ (OPC : 1 : available for OPC-clients) *)		(*Valeur de la consigne de pression ou position demandée*)
	STATE_Mode:					BOOL;	(* ~ (OPC : 1 : available for OPC-clients) *)		(*Mode de régulation en cours*)

	AUTOR_On_IHM:				BOOL; 	(* ~ (OPC : 1 : available for OPC-clients) *)		(*etat ouverture autorisée depuis la supervision en mode manuel*)
	AUTOR_Off_IHM:				BOOL; 	(* ~ (OPC : 1 : available for OPC-clients) *)		(*etat fermeture autorisée depuis la supervision en mode manuel*)
	AUTOR_Lam_IHM:				BOOL;	(* ~ (OPC : 1 : available for OPC-clients) *)		(*etat laminage autorisée depuis la supervision en mode manuel*)
	AUTOR_On_PLC:				BOOL;											(*etat ouverture autorisée depuis l'automate*)
	AUTOR_Off_PLC:				BOOL;											(*etat fermeture autorisée depuis l'automate*)
END_VAR


VAR
	(*retours vanne ouvrete fermée selon retour position*)
	VAR_IN_OFF:					BOOL; 	(* retour vanne fermée*)
	VAR_IN_ON:					BOOL; 	(*retour vanne ouverte*)

	TIMER_Valid_On:				TON;
	TIMER_Valid_Off:			TON;
	TIMER_Valid_Pos_ok:			TON;
	TIMER_Valid_Press_ok:		TON;

	M_On:  						BOOL; 	(* ~ (OPC : 1 : available for OPC-clients) *)		(*Ordre mode manuel ouverture de la vanne*)
	M_Off:   					BOOL; 	(* ~ (OPC : 1 : available for OPC-clients) *)		(*Ordre mode manuel fermeture de la vanne*)
	M_Lam:   					BOOL; 	(* ~ (OPC : 1 : available for OPC-clients) *)		(*Ordre mode manuel de mise en position laminage*)
	RCP_M_On:   				BOOL;
	RCP_M_Off:  				BOOL;
	RCP_M_Lam:					BOOL;
	VAR_On:						BOOL;											(*bit intermédiaire de demande d'ouverture de la vanne*)
	VAR_Lam:					BOOL;											(*bit intermédiaire de demande de mise en laminage de la vanne*)
	VAR_Mem_PRM_Pression:		REAL;											(*variable de mémorisation de la consigne de pression*)
	VAR_Prm_Pression_modifie:	BOOL;											(*variable activée à chaque changement de consigne de pression*)
	VAR_Attente_Stab:			BOOL;											(*variable activée aprés chaque demande de changement de consigne lorsque
																				la stabilisation de pression est attendue*)
	VAR_Surv_Pression:			BOOL;											(*variable indiquant que la pression doit être surveillée - stabilisation atteinte*)
END_VAR

VAR_EXTERNAL
	MANUAL_SAFETY_OFF:		BOOL;											(*desactive les sécurités en mode manuel*)
END_VAR

DEF_On.IdXml					:=	'3';
DEF_On.TagXml					:=	2;

DEF_Off.IdXml					:=	'3';
DEF_Off.TagXml					:=	4;

DEF_On_Imposs.IdXml				:=	'3';
DEF_On_Imposs.TagXml			:=	7;

DEF_Off_Imposs.IdXml			:=	'3';
DEF_Off_Imposs.TagXml			:=	9;

DEF_Off_auto.IdXml				:=	'3';
DEF_Off_auto.TagXml				:=	11;

DEF_Position.IdXml				:=	'16';
DEF_Position.TagXml				:=	9;

DEF_Pression.IdXml				:=	'16';
DEF_Pression.TagXml				:=	8;

DEF_Surv_Pression.IdXml			:=	'16';
DEF_Surv_Pression.TagXml		:=	11;

ALA_Surv_Pression.IdXml			:=	'16';
ALA_Surv_Pression.TagXml		:=	10;
ALA_Surv_Pression.Groupe		:=	1;

(*Traitement du signal d'entrée de position codé sur 100 000 points pour 100%*)
STATE_Position	:=	DINT_TO_REAL(IN_POSITION / 1000);
(*Envoi de la pression de la jauge vers la vanne*)
OUT_Pressure	:=	REAL_TO_DINT(I_PRESSION * 1000000 / CONF_Pr_Max_SP);


(*Mémorisation de la consigne et détection de changement de consigne*)
VAR_Prm_Pression_modifie :=  (PRM_Pression <> VAR_Mem_PRM_pression) AND VAR_Lam AND PRM_MODE AND NOT MANUAL AND NOT RESET;;
IF VAR_Lam AND PRM_mode THEN
	VAR_Mem_PRM_Pression	:= PRM_Pression;
ELSE
	VAR_Mem_PRM_Pression := 0.0;
END_IF;
(*positionnement du bit d'attente de la stabilisation de pression aprés modification de la consigne de pression*)
IF VAR_Prm_Pression_modifie AND NOT MANUAL AND NOT RESET  THEN
	VAR_Attente_Stab := TRUE;
END_IF;

(* Réception des ordres en mode manuel*)
RCP_M_On 			:=	M_On;
RCP_M_Off			:=	M_Off;
RCP_M_Lam			:=	M_Lam;

(*Autorisation*)
AUTOR_On_IHM		:= 	MANUAL AND ((EN_On_INT AND EN_On_EXT)
						OR MANUAL_SAFETY_OFF) AND NOT RESET AND NOT VAR_On;
AUTOR_Off_IHM		:= 	MANUAL AND ((EN_Off_INT AND EN_Off_EXT)  OR
						MANUAL_SAFETY_OFF) AND NOT RESET AND  (VAR_On OR VAR_Lam);
AUTOR_Lam_IHM	:=	MANUAL AND ((EN_On_INT AND EN_On_EXT)
						OR MANUAL_SAFETY_OFF) AND NOT RESET AND NOT VAR_Lam;
AUTOR_On_PLC		:=	NOT MANUAL AND (EN_On_INT AND EN_On_EXT)
						AND NOT RESET;
AUTOR_Off_PLC		:= 	NOT MANUAL AND (EN_Off_INT AND EN_Off_EXT)
						AND NOT RESET;
(*defaut ouverture ou laminage impossible en mode automatique*)
DEF_On_Imposs.CONDITION:=	(CO_On OR CO_Lam) AND NOT AUTOR_On_PLC AND NOT MANUAL;
DEF_On_Imposs.DELAY := T#0ms;
DEF_On_Imposs();
(*Defaut fermeture impossible en mode automatique*)
DEF_Off_Imposs.CONDITION:=	NOT CO_On AND NOT CO_Lam AND NOT AUTOR_Off_PLC AND NOT MANUAL
							AND (VAR_Lam OR VAR_On);
DEF_Off_Imposs.DELAY := T#0ms;
DEF_Off_Imposs();
(*defaut de fermeture automatique de la vanne*)
DEF_Off_Auto.CONDITION :=             (NOT EN_On_INT OR NOT EN_On_EXT) AND  (VAR_On OR VAR_Lam)
								 AND ((CONF_En_ON=1) OR ((CONF_EN_On=0) AND MANUAL)) AND NOT RESET;
DEF_Off_auto.DELAY:=T#0ms;
DEF_Off_Auto();

(*gestion des sorties*)
IF 		(RCP_M_On AND AUTOR_On_IHM) OR
		(CO_On AND AUTOR_On_PLC) THEN
				VAR_On		:= 	TRUE;
				VAR_Lam	:= 	FALSE;
ELSIF 	(RCP_M_Lam AND AUTOR_Lam_IHM) OR
	    	(CO_Lam AND AUTOR_On_PLC) THEN
				VAR_On		:=	FALSE;
				VAR_LAm	:=	TRUE;
ELSIF 	RESET  OR DEF_Off_Auto.DEF OR
		(RCP_M_Off AND AUTOR_Off_IHM) OR
	    	((NOT CO_Lam AND NOT CO_On) AND AUTOR_Off_PLC) THEN
				VAR_On		:= 	FALSE;
				VAR_Lam	:=	FALSE;
END_IF;

(*Gestion du control mode*)
(*Ouverture vanne*)
IF VAR_ON THEN
	OUT_Control_Mode := 4;
END_IF;
(*fermeture vanne*)
IF NOT Var_Lam AND NOT Var_on THEN
	OUT_Control_Mode := 3;
END_IF;
(*régulation pression*)
IF Var_Lam AND PRM_MODE THEN
	OUT_Control_Mode := 5;
END_IF;
(*régulation position*)
IF Var_Lam AND NOT Prm_mode THEN
	OUT_Control_Mode := 2;
END_IF;


(*------Gestion de la consigne analogique pression ou position-----*)
(*Envoi de la consigne de pression*)
IF 		PRM_Mode AND VAR_Lam THEN
			OUT_Pressure_Setpoint	:=	REAL_TO_DINT(PRM_Pression * 1000000 / CONF_Pr_Max_SP);
			STATE_Mode	:=	TRUE;
(*Envoi de la consigne de position*)
ELSIF 	NOT PRM_Mode AND VAR_Lam THEN
			OUT_Position_Setpoint	:=	REAL_TO_DINT(PRM_Position * 1000);
			STATE_Mode	:=	FALSE;
(*RaZ des consignes*)
ELSIF NOT VAR_Lam	THEN
			OUT_Position_Setpoint	:=	0;
			OUT_Pressure_Setpoint	:=	0;
END_IF;


(*Retour vanne ouverte fermée selon position*)
VAR_IN_OFF := (State_position = 0) ;
VAR_IN_ON := (State_position = 100) ;



(*indicateur actionneur activé STATE_ON*)
TIMER_Valid_On.IN	:=	VAR_ON AND VAR_IN_On;
TIMER_Valid_On(PT:=CONF_Tim_Valid_On);
STATE_ON			:=	TIMER_Valid_On.Q;
(*indicateur actionneur activé STATE_OFF*)
TIMER_Valid_Off.IN	:=	NOT VAR_Lam AND NOT VAR_On AND VAR_IN_off;
TIMER_Valid_Off(PT:=CONF_Tim_Valid_Off);
STATE_Off			:=	TIMER_Valid_Off.Q;
(*indicateur STATE_NOK*)
STATE_Nok			:=	DEF_ON.DEF OR DEF_Off.DEF OR DEF_Off_auto.DEF OR DEF_On_Imposs.DEF OR
						DEF_Off_Imposs.DEF OR DEF_pression.DEF OR DEF_Position.DEF;

(*temporisation de validation de la stabilisation à la consigne de position*)
TIMER_Valid_Pos_OK.IN		:=	VAR_Lam AND NOT PRM_Mode AND(  (ABS(STATE_Position - PRM_position) <= CONF_WPos) OR (CONF_WPos = 0.0));
TIMER_Valid_Pos_OK.PT		:=	CONF_Tim_WPos;
Timer_Valid_pos_OK();
STATE_Pos_OK				:= 	TIMER_Valid_Pos_OK.Q;


(*temporisation de validation de la stabilisation à la consigne de pression*)
TIMER_Valid_Press_OK.IN		:=	VAR_Lam AND PRM_Mode AND (((I_Pression >= PRM_W_Pr_LO) AND (I_Pression <= PRM_W_Pr_HI))
								OR (PRM_Tim_W_Pr = T#0ms))
								AND NOT VAR_Prm_Pression_modifie ;
TIMER_Valid_Press_OK.PT		:=	PRM_Tim_W_Pr;
TIMER_Valid_Press_OK();
STATE_Press_OK				:=	TIMER_Valid_Press_ok.Q;

(*indicateur actionneur activé STATE_LAM*)
STATE_Lam			:=	(VAR_Lam AND PRM_Mode) OR (VAR_LAM AND NOT PRM_Mode AND STATE_Pos_ok);
STATE_Ok  			:= 	STATE_Pos_Ok OR STATE_Press_Ok;

(*positionnement du bit de validation de la surveillance de la pression
si la stabilisation de pression est obtenue*)
IF (VAR_Lam AND PRM_MODE AND STATE_Press_ok) AND NOT MANUAL AND NOT RESET  THEN
	VAR_Surv_Pression :=	TRUE;
END_IF;
(*RAZ du bit d'attente de la stabilisation de pression lorsque l'état de stabilisation pression a été atteint ou
que le mode régulation de pression n'est plus demandé*)
IF (VAR_Attente_stab AND STATE_Press_ok) OR RESET OR NOT (VAR_Lam AND PRM_Mode)  THEN
	VAR_Attente_Stab := FALSE;
END_IF;

(*RAZ du bit de surveillance de la stabilisation si pas en mode régulation de pression ou si un changement de consigne est apparu*)
IF VAR_Prm_Pression_modifie  OR RESET OR NOT (VAR_Lam AND PRM_Mode)  THEN
	VAR_Surv_Pression := FALSE;
END_IF;

(*défaut d'ouverture*)
DEF_On.Condition		:= 	VAR_On AND NOT STATE_On;
DEF_On();
(*défaut de fermeture*)
DEF_Off.Condition		:= 	NOT VAR_on AND NOT VAR_Lam AND NOT STATE_Off;
DEF_Off();
(*défaut d'obtention de la position*)
DEF_Position.Condition	:= 	VAR_Lam AND NOT PRM_Mode AND NOT STATE_Pos_Ok;
DEF_position();
(*défaut d'obtention de la pression - le défaut n'est plus surveillé lorsque l'état STATE_Press_ok a été atteint  et est
surveillé de nouveau aprés un changement de consigne*)
DEF_Pression.Condition	:= 	VAR_Lam AND PRM_Mode AND NOT STATE_Press_Ok AND VAR_Attente_Stab
							AND NOT MANUAL AND NOT RESET;
DEF_Pression(DELAY		:=	PRM_Max_Tim_W);

(*défaut de surveillance de la pression - l'état STATE_Press_Ok est perdu pendant un temps supérieur à PRM_TIM_SURV_PR *)
DEF_Surv_Pression.CONDITION	:=	VAR_Lam AND PRM_Mode AND NOT State_Press_OK AND VAR_Surv_Pression
								AND NOT MANUAL AND NOT RESET;
DEF_Surv_Pression (DELAY:=PRM_Tim_Def_Pr);


(*défaut de surveillance de la pression - l'état STATE_Press_Ok est perdu pendant un temps supérieur à PRM_ALA_SURV_PR*)
ALA_Surv_Pression.CONDITION 	:=	VAR_Lam AND PRM_Mode AND NOT State_Press_OK AND VAR_Surv_Pression
									AND NOT MANUAL AND NOT RESET;
ALA_Surv_Pression (DELAY:=PRM_Tim_Ala_Pr);

(* Reset des ordres *)
IF M_On AND RCP_M_On THEN
	M_On 	:= FALSE;
END_IF;
IF M_Off AND RCP_M_Off THEN
	M_Off		 := FALSE;
END_IF;
IF M_Lam AND RCP_M_Lam THEN
	M_Lam		 := FALSE;
END_IF;

END_FUNCTION_BLOCK

// ---- POUs/Composant/VANNES/BLOCK_VVAT_653_ETHERCAT.TcPOU
FUNCTION_BLOCK BLOCK_VVAT_653_ETHERCAT

(* Gestion d'une vanne asservie VAT interface ethercat*)

(****************historique des versions*****************************)

(* Version 1-0 - BC - VERSION INITIALE AC2000 - aff 13741 à partir du bloc VVAT650 Ethercat*)
(* sur cette version: 
changement de in_position en DINT->real
basé sur 100 points au lieu de 100 000

changement de OUT_Pressure en DINT->real
changement de OUT_Position_Setpoint en DINT->real
changement de OUT_Pressure_Setpoint en DINT->real

*)
(*
Configuration vanne : Startup CoE :
Param 0x20F5 _ valeur 0x02 ==> sensor 1 unit à mbar

Configuration vanne via le logiciel VAT CPA , dans terminal :
envoi de la commande 		a:74031 
Cette commande sert à mettre la réception de la pression jauge sur external digital output sensor 1

envoi de la commande		s:2309000000
Cette commande sert à mettre le signal de reception jauge sur un DINT, range par défaut ==> sans doute inutile de la mettre	

Signal de la jauge process envoyée au bloc par entrée I_Pressure (REAL)
Information pression envoyée à la vanne par OUT_Pression_Ethercat (DINT, avec max range de 1 000 000)*)
(*Version 1-1 - HG - Défauts après gestion des demandes pour éviter le défaut fermeture impossible sur arrêt machine*)

(*************************************************************************)

VAR_INPUT
(*paramètre standard*)
	RESET:   					BOOL; 		(*Condition RAZ actionneur*)
	MANUAL:  					BOOL; 		(*Mode manuel*)

(*entrée externe*)
	IN_OFF:						BOOL; 		(*E.TOR vanne fermée*)
	IN_ON:						BOOL; 		(*E.TOR vanne ouverte*)

	IN_POSITION		AT%I*:		REAL;		(*Retour de position de la jauge, de 0 à 100 points*)
	I_PRESSION:					REAL;		(*Mesure de pression externe*)

(*Paramètres*)
	PRM_Mode:					BOOL; 		(*Mode FALSE = Position / TRUE = Pression*)
	PRM_Pression:				REAL; 		(*Consigne de pression - en unité cohérente avec la mesure*)
	PRM_Position:				REAL;		(*Consigne de position de la vanne en %*)
	PRM_W_Pr_HI:				REAL;		(*Tolérance haute de stabilisation de pression pour obtention de l'état stab pression ok*)
	PRM_W_Pr_LO:				REAL;		(*Tolérance basse de dtabilisation de pression pour obtention de l'état stab pression ok*)
	PRM_Tim_W_Pr:				TIME;		(*Temps de validation de stabilisation de la pression*)

(*défaut du bloc*)
	DEF_On:  					PRCDEF; 	(*00 - Défaut d'ouverture de la vanne*)
	DEF_Off:   					PRCDEF; 	(*01 - Défaut de fermeture de la vanne*)
	DEF_On_Imposs:				PRCDEF;		(*03 - Défaut d'ouverture ou de mise en laminage non autorisée en mode automatique*)
	DEF_Off_Imposs:				PRCDEF;		(*04 - Défaut de fermeture non autorisée en mode automatique*)
	DEF_Off_auto:				PRCDEF;		(*05 - Défaut de fermeture automatique de la vanne*)
	DEF_Position:				PRCDEF;		(*06 - Défaut d'obtention de la position*)
	DEF_Pression:				PRCDEF;		(*07 - Défaut d'obtention de la pression*)
	DEF_Surv_Pression:			PRCDEF;		(*08 - Défaut de surveillance de la pression - perte du critère de stabilisation*)
	ALA_Surv_Pression:			PRCDEF;		(*09 - Alarme de surveillance de la rpession - perte du critère de stabilisation*)

(*parametre de pilotage en entrée*)
	CO_On:   					BOOL;		(*Ordre mode automatique ouverture*)
	CO_Lam:						BOOL;		(*Ordre mode automatique laminage*)
	EN_On_INT:   				BOOL;		(*Condition d'autorisation d'ouverture ou de laminage donnée par le bloc qui instancie le bloc actuator*)
	EN_Off_INT:  				BOOL;		(*Condition d'autorisation de fermeture donnée par le bloc qui instacie le bloc actuator*)
	EN_On_EXT:					BOOL:=TRUE;	(*condition d'autorisation d'ouverture ou de laminage externe*)
	EN_Off_EXT:					BOOL:=TRUE;	(*condition d'autorisation de fermeture externe*)
END_VAR

VAR_OUTPUT
	OUT_Pressure			AT%Q*:	REAL;	(*envoi de la pression reçue par jauge sur trame ethercat, codée sur 1 000 000 point pour pleine échelle*)
	OUT_Control_Mode		AT%Q*:	SINT;	(*control mode : 2-position, 3-close, 4-open, 5-pression*)
	OUT_Pressure_Setpoint	AT%Q*:	REAL;	(*consigne puissance, codé sur 1 000 000 points pour pleine echelle*)
	OUT_Position_Setpoint	AT%Q*:	REAL;	(*consigne position , codé sur 100 000 point pour 100%*)

	STATE_On:	   				BOOL; 		(*Indicateur ouverture ok*)
	STATE_Off:  				BOOL; 		(*Indicateur fermeture ok*)
	STATE_Nok:					BOOL;		(*Indicateur défaut sur la vanne*)
	STATE_Lam:					BOOL;		(*Indicateur mise en laminage ok *)
	STATE_Pos_Ok:				BOOL;		(*Indicateur de positionnement de la vanne ok *)
	STATE_Press_Ok:				BOOL;		(*Indicateur de stabilisation de la pression ok *)
	STATE_Ok:					BOOL;		(*Indicateur de stabilisation autour du point de consigne de pression
												ou de positionnement ok si le controle est en mode position*)
	STATE_Position:				REAL;		(*Retour de position de la vanne*)
	STATE_Setpoint:				REAL;		(*Valeur de la consigne de pression ou position demandée*)
	STATE_Mode:					BOOL;		(*Mode de régulation en cours*)

	AUTOR_On_IHM:				BOOL; 		(*etat ouverture autorisée depuis la supervision en mode manuel*)
	AUTOR_Off_IHM:				BOOL; 		(*etat fermeture autorisée depuis la supervision en mode manuel*)
	AUTOR_Lam_IHM:				BOOL;		(*etat laminage autorisée depuis la supervision en mode manuel*)
	AUTOR_On_PLC:				BOOL;		(*etat ouverture autorisée depuis l'automate*)
	AUTOR_Off_PLC:				BOOL;		(*etat fermeture autorisée depuis l'automate*)
END_VAR

VAR
	(*retours vanne ouvrete fermée selon retour position*)
	VAR_IN_OFF:					BOOL; 		(* retour vanne fermée*)
	VAR_IN_ON:					BOOL; 		(*retour vanne ouverte*)

	TIMER_Valid_On:				TON;
	TIMER_Valid_Off:			TON;
	TIMER_Valid_Pos_ok:			TON;
	TIMER_Valid_Press_ok:		TON;

	M_On:  						BOOL; 		(*Ordre mode manuel ouverture de la vanne*)
	M_Off:   					BOOL; 		(*Ordre mode manuel fermeture de la vanne*)
	M_Lam:   					BOOL; 		(*Ordre mode manuel de mise en position laminage*)
	RCP_M_On:   				BOOL;
	RCP_M_Off:  				BOOL;
	RCP_M_Lam:					BOOL;
	VAR_On:						BOOL;		(*bit intermédiaire de demande d'ouverture de la vanne*)
	VAR_Lam:					BOOL;		(*bit intermédiaire de demande de mise en laminage de la vanne*)
	VAR_Mem_PRM_Pression:		REAL;		(*variable de mémorisation de la consigne de pression*)
	VAR_Prm_Pression_modifie:	BOOL;		(*variable activée à chaque changement de consigne de pression*)
	VAR_Attente_Stab:			BOOL;		(*variable activée aprés chaque demande de changement de consigne lorsque
												la stabilisation de pression est attendue*)
	VAR_Surv_Pression:			BOOL;		(*variable indiquant que la pression doit être surveillée - stabilisation atteinte*)
END_VAR

VAR_INPUT PERSISTENT
	(*Entité*)
	IsComponent:				BOOL;		(*entité : composant*)
	IdXML:						STRING;		(*nom entité : identifiant pour recherche dans dico*)
	TagXML:						UINT;		(*nom entité : identifiant pour recherche dans dico*)
	IdParent:					STRING;		(*MNEMO de l'appelant*)
	MNEMO:						STRING;		(*MNEMO de l'entité*)

(*parametre de configuration constructeur*)
(*les parametres suivants dépendent de la configuration de la machine*)
	CONF_Tim_Valid_On:  		TIME:=T#100MS; 	(*Temps validation de la position ouverte *)
	CONF_Tim_Valid_Off:   		TIME:=T#100MS; 	(*Temps validation de la position fermée *)
	CONF_EN_On:					USINT:=0;		(*définit la réaction du système en cas de perte des conditions d'autorisation d'activation EN_On*)
													(* 0 = désactivation automatique  en cas de perte des conditions d'autorisation d'activation uniquement en manuel*)
													(* 1 = désactivation automatique en cas de perte des conditions d'autorisation d'activation en auto et en manuel*)
													(* 2 = Pas de déscativation automatique*)
	CONF_Pr_Max_SP:				REAL;			(* Consigne max. de pression en pleine echelle 10V - correspond à la pleine échelle du capteur connecté au coffret*)
	CONF_WPos:					REAL;			(*Tolérance de positionnement pour obtention de l'état STATE_POS_ok*)
	CONF_Tim_WPos:				TIME;			(*Temps de validation de l'état STATE_POS_Ok*)
	PRM_Max_Tim_W:				TIME;			(*Temps Max d'obtention de l'état stabilisation pression ok*)
	PRM_Tim_Def_Pr:				TIME;			(*Temps d'enveloppe du défaut de surveillance de la pression*)
	PRM_Tim_Ala_Pr:				TIME;			(*Temps d'enveloppe de l'alarme de surveillance de la pression*)
END_VAR

DEF_On.IdXml					:=	'3';
DEF_On.TagXml					:=	2;

DEF_Off.IdXml					:=	'3';
DEF_Off.TagXml					:=	4;

DEF_On_Imposs.IdXml				:=	'3';
DEF_On_Imposs.TagXml			:=	7;

DEF_Off_Imposs.IdXml				:=	'3';
DEF_Off_Imposs.TagXml			:=	9;

DEF_Off_auto.IdXml				:=	'3';
DEF_Off_auto.TagXml				:=	11;

DEF_Position.IdXml				:=	'1';
DEF_Position.TagXml				:=	9;

DEF_Pression.IdXml				:=	'1';
DEF_Pression.TagXml				:=	8;

DEF_Surv_Pression.IdXml			:=	'1';
DEF_Surv_Pression.TagXml		:=	11;

ALA_Surv_Pression.IdXml			:=	'1';
ALA_Surv_Pression.TagXml		:=	10;
ALA_Surv_Pression.Groupe		:=	1;

(*Traitement du signal d'entrée de position codé sur 100 000 points pour 100%*)
STATE_Position	:=	IN_POSITION;
(*Envoi de la pression de la jauge vers la vanne*)
OUT_Pressure	:=	I_PRESSION;//* 1000000 / CONF_Pr_Max_SP);


(*Mémorisation de la consigne et détection de changement de consigne*)
VAR_Prm_Pression_modifie :=  (PRM_Pression <> VAR_Mem_PRM_pression) AND VAR_Lam AND PRM_MODE AND NOT MANUAL AND NOT RESET;;
IF VAR_Lam AND PRM_mode THEN
	VAR_Mem_PRM_Pression	:= PRM_Pression;
ELSE
	VAR_Mem_PRM_Pression 	:= 0.0;
END_IF;
(*positionnement du bit d'attente de la stabilisation de pression aprés modification de la consigne de pression*)
IF VAR_Prm_Pression_modifie AND NOT MANUAL AND NOT RESET  THEN
	VAR_Attente_Stab 		:= TRUE;
END_IF;

(* Réception des ordres en mode manuel*)
RCP_M_On 			:=	M_On;
RCP_M_Off			:=	M_Off;
RCP_M_Lam			:=	M_Lam;

(*Autorisation*)
AUTOR_On_IHM		:= 	MANUAL AND ((EN_On_INT AND EN_On_EXT)
						OR MANUAL_SAFETY_OFF) AND NOT RESET AND NOT VAR_On;
AUTOR_Off_IHM		:= 	MANUAL AND ((EN_Off_INT AND EN_Off_EXT)  OR
						MANUAL_SAFETY_OFF) AND NOT RESET AND  (VAR_On OR VAR_Lam);
AUTOR_Lam_IHM		:=	MANUAL AND ((EN_On_INT AND EN_On_EXT)
						OR MANUAL_SAFETY_OFF) AND NOT RESET AND NOT VAR_Lam;
AUTOR_On_PLC		:=	NOT MANUAL AND (EN_On_INT AND EN_On_EXT)
						AND NOT RESET;
AUTOR_Off_PLC		:= 	NOT MANUAL AND (EN_Off_INT AND EN_Off_EXT)
						AND NOT RESET;

(*gestion des sorties*)
IF 		(RCP_M_On AND AUTOR_On_IHM) OR
		(CO_On AND AUTOR_On_PLC) THEN
				VAR_On		:= 	TRUE;
				VAR_Lam		:= 	FALSE;
ELSIF 	(RCP_M_Lam AND AUTOR_Lam_IHM) OR
	    (CO_Lam AND AUTOR_On_PLC) THEN
				VAR_On		:=	FALSE;
				VAR_LAm		:=	TRUE;
ELSIF 	RESET  OR DEF_Off_Auto.DEF OR
		(RCP_M_Off AND AUTOR_Off_IHM) OR
	    ((NOT CO_Lam AND NOT CO_On) AND AUTOR_Off_PLC) THEN
				VAR_On		:= 	FALSE;
				VAR_Lam		:=	FALSE;
END_IF;

(*defaut ouverture ou laminage impossible en mode automatique*)
DEF_On_Imposs.CONDITION	:=	(CO_On OR CO_Lam) AND NOT AUTOR_On_PLC AND NOT MANUAL;
DEF_On_Imposs.DELAY 	:= 	T#0MS;
DEF_On_Imposs();
(*Defaut fermeture impossible en mode automatique*)
DEF_Off_Imposs.CONDITION:=	NOT CO_On AND NOT CO_Lam AND NOT AUTOR_Off_PLC AND NOT MANUAL
							AND (VAR_Lam OR VAR_On);
DEF_Off_Imposs.DELAY 	:= 	T#0MS;
DEF_Off_Imposs();
(*defaut de fermeture automatique de la vanne*)
DEF_Off_Auto.CONDITION 	:=	(NOT EN_On_INT OR NOT EN_On_EXT) AND (VAR_On OR VAR_Lam)
							AND ((CONF_En_ON=1) OR ((CONF_EN_On=0) AND MANUAL)) AND NOT RESET;
DEF_Off_auto.DELAY:=T#0ms;
DEF_Off_Auto();

(*Gestion du control mode*)
(*Ouverture vanne*)
IF VAR_ON THEN
	OUT_Control_Mode := 4;
END_IF;
(*fermeture vanne*)
IF NOT Var_Lam AND NOT Var_on THEN
	OUT_Control_Mode := 3;
END_IF;
(*régulation pression*)
IF Var_Lam AND PRM_MODE THEN
	OUT_Control_Mode := 5;
END_IF;
(*régulation position*)
IF Var_Lam AND NOT Prm_mode THEN
	OUT_Control_Mode := 2;
END_IF;


(*------Gestion de la consigne analogique pression ou position-----*)
(*Envoi de la consigne de pression*)
IF	PRM_Mode AND VAR_Lam THEN
	OUT_Pressure_Setpoint	:=	PRM_Pression;// * 1000000 / CONF_Pr_Max_SP);
	STATE_Mode				:=	TRUE;
(*Envoi de la consigne de position*)
ELSIF NOT PRM_Mode AND VAR_Lam THEN
	OUT_Position_Setpoint	:=	PRM_Position;// * 1000;
	STATE_Mode				:=	FALSE;
(*RaZ des consignes*)
ELSIF NOT VAR_Lam	THEN
	OUT_Position_Setpoint	:=	0;
	OUT_Pressure_Setpoint	:=	0;
END_IF;

(*Retour vanne ouverte fermée selon position*)
VAR_IN_OFF 	:=	(State_position = 0) ;
VAR_IN_ON	:= 	(State_position = 100) ;

(*indicateur actionneur activé STATE_ON*)
TIMER_Valid_On.IN	:=	VAR_ON AND VAR_IN_On;
TIMER_Valid_On(PT:=CONF_Tim_Valid_On);
STATE_ON			:=	TIMER_Valid_On.Q;
(*indicateur actionneur activé STATE_OFF*)
TIMER_Valid_Off.IN	:=	NOT VAR_Lam AND NOT VAR_On AND VAR_IN_off;
TIMER_Valid_Off(PT:=CONF_Tim_Valid_Off);
STATE_Off			:=	TIMER_Valid_Off.Q;
(*indicateur STATE_NOK*)
STATE_Nok			:=	DEF_ON.DEF OR DEF_Off.DEF OR DEF_Off_auto.DEF OR DEF_On_Imposs.DEF OR
						DEF_Off_Imposs.DEF OR DEF_pression.DEF OR DEF_Position.DEF;

(*temporisation de validation de la stabilisation à la consigne de position*)
TIMER_Valid_Pos_OK.IN		:=	VAR_Lam AND NOT PRM_Mode AND(  (ABS(STATE_Position - PRM_position) <= CONF_WPos) OR (CONF_WPos = 0.0));
TIMER_Valid_Pos_OK.PT		:=	CONF_Tim_WPos;
Timer_Valid_pos_OK();
STATE_Pos_OK				:= 	TIMER_Valid_Pos_OK.Q;


(*temporisation de validation de la stabilisation à la consigne de pression*)
TIMER_Valid_Press_OK.IN		:=	VAR_Lam
								AND PRM_Mode
								AND (((I_Pression >= PRM_W_Pr_LO)
									AND (I_Pression <= PRM_W_Pr_HI))
											OR (PRM_Tim_W_Pr = T#0ms))
								AND NOT VAR_Prm_Pression_modifie ;
TIMER_Valid_Press_OK.PT	:=	PRM_Tim_W_Pr;
TIMER_Valid_Press_OK();
STATE_Press_OK			:=	TIMER_Valid_Press_ok.Q;

(*indicateur actionneur activé STATE_LAM*)
STATE_Lam	:=	(VAR_Lam AND PRM_Mode) OR (VAR_LAM AND NOT PRM_Mode AND STATE_Pos_ok);
STATE_Ok  	:= 	STATE_Pos_Ok OR STATE_Press_Ok;

(*positionnement du bit de validation de la surveillance de la pression
si la stabilisation de pression est obtenue*)
IF (VAR_Lam AND PRM_MODE AND STATE_Press_ok) AND NOT MANUAL AND NOT RESET  THEN
	VAR_Surv_Pression :=	TRUE;
END_IF;
(*RAZ du bit d'attente de la stabilisation de pression lorsque l'état de stabilisation pression a été atteint ou
que le mode régulation de pression n'est plus demandé*)
IF (VAR_Attente_stab AND STATE_Press_ok) OR RESET OR NOT (VAR_Lam AND PRM_Mode)  THEN
	VAR_Attente_Stab := FALSE;
END_IF;

(*RAZ du bit de surveillance de la stabilisation si pas en mode régulation de pression ou si un changement de consigne est apparu*)
IF VAR_Prm_Pression_modifie  OR RESET OR NOT (VAR_Lam AND PRM_Mode)  THEN
	VAR_Surv_Pression := FALSE;
END_IF;

(*défaut d'ouverture*)
DEF_On.Condition			:= 	VAR_On AND NOT STATE_On;
DEF_On();
(*défaut de fermeture*)
DEF_Off.Condition			:= 	NOT VAR_on AND NOT VAR_Lam AND NOT STATE_Off;
DEF_Off();
(*défaut d'obtention de la position*)
DEF_Position.Condition	:= 	VAR_Lam AND NOT PRM_Mode AND NOT STATE_Pos_Ok;
DEF_position();
(*défaut d'obtention de la pression - le défaut n'est plus surveillé lorsque l'état STATE_Press_ok a été atteint  et est
surveillé de nouveau aprés un changement de consigne*)
DEF_Pression.Condition	:= 	VAR_Lam
							AND PRM_Mode
							AND NOT STATE_Press_Ok
							AND VAR_Attente_Stab
							AND NOT MANUAL
							AND NOT RESET;
DEF_Pression(DELAY		:=	PRM_Max_Tim_W);

(*défaut de surveillance de la pression - l'état STATE_Press_Ok est perdu pendant un temps supérieur à PRM_TIM_SURV_PR *)
DEF_Surv_Pression.CONDITION	:=	VAR_Lam
								AND PRM_Mode
								AND NOT ((I_Pression >= PRM_W_Pr_LO)
									AND (I_Pression <= PRM_W_Pr_HI))
								AND VAR_Surv_Pression
								AND NOT MANUAL
								AND NOT RESET;
DEF_Surv_Pression (DELAY:=PRM_Tim_Def_Pr);

(*défaut de surveillance de la pression - l'état STATE_Press_Ok est perdu pendant un temps supérieur à PRM_ALA_SURV_PR*)
ALA_Surv_Pression.CONDITION 	:=	VAR_Lam
									AND PRM_Mode
									AND NOT ((I_Pression >= PRM_W_Pr_LO)
										AND (I_Pression <= PRM_W_Pr_HI))
									AND VAR_Surv_Pression
									AND NOT MANUAL
									AND NOT RESET;
ALA_Surv_Pression (DELAY:=PRM_Tim_Ala_Pr);

(* Reset des ordres *)
IF M_On AND RCP_M_On THEN
	M_On 	:= FALSE;
END_IF;
IF M_Off AND RCP_M_Off THEN
	M_Off	:= FALSE;
END_IF;
IF M_Lam AND RCP_M_Lam THEN
	M_Lam	:= FALSE;
END_IF;

END_FUNCTION_BLOCK

// ---- POUs/FONCTION DE BASE/Format String/FORMAT_FLOAT_STRING.TcPOU
FUNCTION FORMAT_FLOAT_STRING : STRING
VAR_INPUT
	IN_REAL:					REAL;
	NB_DEC_APRES_SEPARATEUR:	INT;
	OP_EXP:						BOOL;
END_VAR
VAR
	VAR_String:		STRING;
	VAR_String2:	STRING;
	VAR_I:			INT;
	VAR_J:			INT;
	VAR_K:			INT;
	VAR_Point:		BOOL;
	VAR_Entier:		BOOL;
END_VAR

(*conversion réel en string*)
VAR_String	:=	REAL_TO_STRING(IN_REAL);

(*recherche exposant*)
VAR_J 	:=	FIND(VAR_String,'E');
(*si format déjà en exposant, fonction terminée*)
IF VAR_J > 0 THEN
	FORMAT_FLOAT_STRING	:=	VAR_String;
	RETURN;
END_IF

(*recherche emplacement séparateur décimal*)
VAR_J	:=	FIND(VAR_String,'.');
IF VAR_J = 0 THEN
	VAR_J		:=	FIND(VAR_String,',');
	VAR_Point	:=	FALSE;
ELSE
	VAR_Point	:=	TRUE;
END_IF

(*longueur chaine initiale*)
VAR_I	:=	LEN(VAR_String);

(*format pas exponentiel ou format exponentiel mais chiffre avant le séparateur décimal*)
VAR_String2	:=	LEFT(VAR_String,1);

IF NOT OP_EXP OR (OP_EXP AND STRING_TO_INT(VAR_String2) > 0) THEN
	(*nombre de caractères à conserver*)
	IF NB_DEC_APRES_SEPARATEUR > 0 THEN
		VAR_K 	:= 	VAR_J + NB_DEC_APRES_SEPARATEUR; 
	ELSE
		VAR_K 	:=	VAR_J - 1; 
	END_IF
	(*chaine de sortie*)
	FORMAT_FLOAT_STRING	:=	LEFT(VAR_String,VAR_K);

ELSE

	(*suppression des chiffres avant le séparateur et le séparateur*)
	VAR_String	:=	RIGHT(VAR_String,VAR_I - VAR_J);
	VAR_I		:=	LEN(VAR_String);
	
	(*suprresion des zeros à gauche*)
	VAR_K := 1;
	VAR_String2 	:= 	MID(VAR_String,1,VAR_K);
	IF VAR_String2 <> '0' THEN
		VAR_K  		:= 	0;
	ELSE
		WHILE (VAR_K <= VAR_I) AND (VAR_String2 = '0') DO
			 VAR_String2 	:= 	MID(VAR_String,1,VAR_K);
			 VAR_K			:=	VAR_K + 1;
		END_WHILE	
		VAR_K  		:= 	VAR_K - 2;
		VAR_String 	:= 	RIGHT(VAR_String,VAR_I-VAR_K);
	END_IF
	
	(*récupération du premier chiffre a supprimer pour arrondir si nécessaire*)
	VAR_I		:=	LEN(VAR_String);
	(*si chaine plus longue que nécessaire*)
	IF VAR_I > NB_DEC_APRES_SEPARATEUR + 1 THEN
		VAR_J := STRING_TO_INT(MID(VAR_String,1,NB_DEC_APRES_SEPARATEUR+2));
		IF  VAR_J >= 5 THEN
			VAR_J := STRING_TO_INT(MID(VAR_String,1,NB_DEC_APRES_SEPARATEUR+1));
			VAR_J := VAR_J + 1;
			VAR_String	:=	CONCAT(LEFT(VAR_String,NB_DEC_APRES_SEPARATEUR),INT_TO_STRING(VAR_J));
		ELSE
			VAR_String	:=	LEFT(VAR_String,NB_DEC_APRES_SEPARATEUR+1);
		END_IF
		(*ajout zéro si chaine pas assez longue*)
	ELSE
		FOR VAR_J := 1 TO NB_DEC_APRES_SEPARATEUR + 1 - VAR_I DO
			VAR_String	:=	CONCAT(VAR_String,'0');
		END_FOR
	END_IF
	
	(*rajout séparateur*)
	IF VAR_Point THEN
		VAR_String	:=	INSERT(VAR_String,'.',1);
	ELSE
		VAR_String	:=	INSERT(VAR_String,',',1);
	END_IF
	
	(*rajout e-*)
	VAR_String	:=	CONCAT(VAR_String,'E-');
	
	(*rajout expostant*)
	VAR_String			:=	CONCAT(VAR_String,INT_TO_STRING(VAR_K+1));
	FORMAT_FLOAT_STRING	:=	VAR_String;
	
END_IF

END_FUNCTION

// ---- POUs/FONCTION DE BASE/IEEE754_INPUT.TcPOU
FUNCTION_BLOCK IEEE754_INPUT

(*fonction de conversion de trame de type IEEE754 (4 octets) en réel simple précision*)

VAR_INPUT
 	INPUT:				ARRAY[0..3] OF USINT;					(*trame d'entrée*)
END_VAR

VAR_OUTPUT
	Value:				REAL;								(*value convertie*)
END_VAR

VAR
	VAR_calcul_entree:	DINT;
	VAR_signe:			INT;
	VAR_calcul_exposant:INT;
	VAR_exposant:		INT;
	VAR_mantisse:		REAL;
END_VAR

(*calcul de la pression*)
VAR_calcul_entree.0 := INPUT[0].0;
VAR_calcul_entree.1 := INPUT[0].1;
VAR_calcul_entree.2 := INPUT[0].2;
VAR_calcul_entree.3 := INPUT[0].3;
VAR_calcul_entree.4 := INPUT[0].4;
VAR_calcul_entree.5 := INPUT[0].5;
VAR_calcul_entree.6 := INPUT[0].6;
VAR_calcul_entree.7 := INPUT[0].7;

VAR_calcul_entree.8 := INPUT[1].0;
VAR_calcul_entree.9 := INPUT[1].1;
VAR_calcul_entree.10 := INPUT[1].2;
VAR_calcul_entree.11 := INPUT[1].3;
VAR_calcul_entree.12 := INPUT[1].4;
VAR_calcul_entree.13 := INPUT[1].5;
VAR_calcul_entree.14 := INPUT[1].6;
VAR_calcul_entree.15 := INPUT[1].7;

VAR_calcul_entree.16 := INPUT[2].0;
VAR_calcul_entree.17 := INPUT[2].1;
VAR_calcul_entree.18 := INPUT[2].2;
VAR_calcul_entree.19 := INPUT[2].3;
VAR_calcul_entree.20 := INPUT[2].4;
VAR_calcul_entree.21 := INPUT[2].5;
VAR_calcul_entree.22 := INPUT[2].6;
VAR_calcul_entree.23 := INPUT[2].7;

VAR_calcul_entree.24 := INPUT[3].0;
VAR_calcul_entree.25 := INPUT[3].1;
VAR_calcul_entree.26 := INPUT[3].2;
VAR_calcul_entree.27 := INPUT[3].3;
VAR_calcul_entree.28 := INPUT[3].4;
VAR_calcul_entree.29 := INPUT[3].5;
VAR_calcul_entree.30 := INPUT[3].6;
VAR_calcul_entree.31 := INPUT[3].7;

IF INPUT[0]<>0OR INPUT[1]<>0OR INPUT[2]<>0 THEN

VAR_signe := BOOL_TO_INT(VAR_calcul_entree.31);

VAR_calcul_exposant.7 := VAR_calcul_entree.30;
VAR_calcul_exposant.6 := VAR_calcul_entree.29;
VAR_calcul_exposant.5 := VAR_calcul_entree.28;
VAR_calcul_exposant.4 := VAR_calcul_entree.27;
VAR_calcul_exposant.3 := VAR_calcul_entree.26;
VAR_calcul_exposant.2 := VAR_calcul_entree.25;
VAR_calcul_exposant.1 := VAR_calcul_entree.24;
VAR_calcul_exposant.0 := VAR_calcul_entree.23;

VAR_exposant := VAR_calcul_exposant - 127;

VAR_mantisse :=	1* EXPT(2,0)
				+ BOOL_TO_INT(VAR_calcul_entree.22) * EXPT(2,-1)
				+ BOOL_TO_INT(VAR_calcul_entree.21) * EXPT(2,-2)
				+ BOOL_TO_INT(VAR_calcul_entree.20) * EXPT(2,-3)
				+ BOOL_TO_INT(VAR_calcul_entree.19) * EXPT(2,-4)
				+ BOOL_TO_INT(VAR_calcul_entree.18) * EXPT(2,-5)
				+ BOOL_TO_INT(VAR_calcul_entree.17) * EXPT(2,-6)
				+ BOOL_TO_INT(VAR_calcul_entree.16) * EXPT(2,-7)
				+ BOOL_TO_INT(VAR_calcul_entree.15) * EXPT(2,-8)
				+ BOOL_TO_INT(VAR_calcul_entree.14) * EXPT(2,-9)
				+ BOOL_TO_INT(VAR_calcul_entree.13) * EXPT(2,-10)
				+ BOOL_TO_INT(VAR_calcul_entree.12) * EXPT(2,-11)
				+ BOOL_TO_INT(VAR_calcul_entree.11) * EXPT(2,-12)
				+ BOOL_TO_INT(VAR_calcul_entree.10) * EXPT(2,-13)
				+ BOOL_TO_INT(VAR_calcul_entree.9) * EXPT(2,-14)
				+ BOOL_TO_INT(VAR_calcul_entree.8) * EXPT(2,-15)
				+ BOOL_TO_INT(VAR_calcul_entree.7) * EXPT(2,-16)
				+ BOOL_TO_INT(VAR_calcul_entree.6) * EXPT(2,-17)
				+ BOOL_TO_INT(VAR_calcul_entree.5) * EXPT(2,-18)
				+ BOOL_TO_INT(VAR_calcul_entree.4) * EXPT(2,-19)
				+ BOOL_TO_INT(VAR_calcul_entree.3) * EXPT(2,-20)
				+ BOOL_TO_INT(VAR_calcul_entree.2) * EXPT(2,-21)
				+ BOOL_TO_INT(VAR_calcul_entree.1) * EXPT(2,-22)
				+ BOOL_TO_INT(VAR_calcul_entree.0) * EXPT(2,-23);

Value := EXPT(-1,Var_signe) * VAR_mantisse * EXPT(2,VAR_exposant);
ELSE
	Value:= 0;
END_IF

END_FUNCTION_BLOCK

// ---- POUs/FONCTION DE BASE/IEEE754_OUTPUT.TcPOU
FUNCTION_BLOCK IEEE754_OUTPUT

(*fonction de conversion de trame de type IEEE754 (4 octets) en réel simple précision*)

VAR_INPUT
	IN_Value:				REAL;								(*valeur a convertir*)
END_VAR

VAR_OUTPUT
	OUTPUT:				ARRAY[0..3] OF USINT;					(*trame de sortie*)
END_VAR

VAR
	VAR_valeur_entiere:			DINT; 		(*valeur entiere du reel a convertir*)
	VAR_value2:			DWORD;
	VAR_valeur_decimal:			REAL;		(*partie decimal de la valeur a convertir*)
	VAR_value_entiere_corrige:	DINT;
	Var_value_corrige:	REAL;
	VAR_calcul_mantisse_temp:	DINT;
	VAR_calcul_mantisse_temp2:	DWORD;
	VAR_signe:			BOOL;
	VAR_calcul_exposant:	INT;
	VAR_exposant:		INT;
	VAR_mantisse:		REAL;
	VAR_mantisse2:		ARRAY[0..32]	OF REAL;
	VAR_CALCUL_SORTIE: DINT;
	I:		INT;
	J:		BYTE;
	N:		BYTE;
	Var_decalage_bit:	BYTE;
	VAR_mantisse_decimal: DWORD;
	VAR_mantisse_entier: DWORD;
	VAR_mantisse_final: DWORD;
	VAR_mantisse_final2: DWORD;
	VAR_nb_zero: INT;
END_VAR

(*calcul de la pression*)

IF IN_Value<0 THEN
	VAR_SIGNE:=TRUE;
ELSIF IN_Value>0 THEN
	VAR_SIGNE:=FALSE;
ELSIF IN_Value= 0 THEN
	VAR_SIGNE:=FALSE;
END_IF

VAR_valeur_entiere:= ABS(REAL_TO_DINT (IN_Value));
VAR_valeur_decimal := ABS(IN_Value) - VAR_valeur_entiere;

IF VAR_valeur_decimal < 0 THEN
Var_value_corrige := 1+ VAR_valeur_decimal;
VAR_value_entiere_corrige:=VAR_valeur_entiere -1;
ELSE Var_value_corrige := VAR_valeur_decimal;
	VAR_value_entiere_corrige:=VAR_valeur_entiere;
END_IF

VAR_calcul_mantisse_temp:=0;
I:=0;

VAR_mantisse2[0]:= Var_value_corrige;

FOR I:=1 TO 32 DO

VAR_mantisse2[I]:= VAR_mantisse2[I-1]*2;

IF VAR_mantisse2[1] >1 THEN
VAR_calcul_mantisse_temp.31:=TRUE;
VAR_mantisse2[1]:= VAR_mantisse2[1] -1;
ELSIF VAR_mantisse2[1] =1 THEN
VAR_calcul_mantisse_temp.31:=TRUE;
VAR_mantisse2[2]:=0;
VAR_mantisse2[3]:=0;
VAR_mantisse2[4]:=0;
VAR_mantisse2[5]:=0;
VAR_mantisse2[6]:=0;
VAR_mantisse2[7]:=0;
VAR_mantisse2[8]:=0;
VAR_mantisse2[9]:=0;
VAR_mantisse2[10]:=0;
VAR_mantisse2[11]:=0;
VAR_mantisse2[12]:=0;
VAR_mantisse2[13]:=0;
VAR_mantisse2[14]:=0;
VAR_mantisse2[15]:=0;
VAR_mantisse2[16]:=0;
VAR_mantisse2[17]:=0;
VAR_mantisse2[18]:=0;
VAR_mantisse2[19]:=0;
VAR_mantisse2[20]:=0;
VAR_mantisse2[21]:=0;
VAR_mantisse2[22]:=0;
VAR_mantisse2[23]:=0;
VAR_mantisse2[24]:=0;
VAR_mantisse2[25]:=0;
VAR_mantisse2[26]:=0;
VAR_mantisse2[27]:=0;
VAR_mantisse2[28]:=0;
VAR_mantisse2[29]:=0;
VAR_mantisse2[30]:=0;
VAR_mantisse2[31]:=0;
VAR_mantisse2[32]:=0;
END_IF;

